    !Tr_meulage_motif_2 : Meulage d'un motif
    LOCAL CONST Robtarget Tr_meulage_motif_2_0 := [[50.49266796875,-116.5996484375,2.28227856445312],[0.000687502564593619,0.0161290141827085,0.042580986650659,-0.998962582791555],[0,0,0,0],[8.999999E+09,8.999999E+09,8.999999E+09,8.999999E+09,8.999999E+09,8.999999E+09]];
    LOCAL CONST Robtarget Tr_meulage_motif_2_1 := [[51.49176171875,-116.5571171875,2.28183227539063],[0.000687502564593619,0.0161290141827085,0.042580986650659,-0.998962582791555],[0,0,0,0],[8.999999E+09,8.999999E+09,8.999999E+09,8.999999E+09,8.999999E+09,8.999999E+09]];
    LOCAL CONST Robtarget Tr_meulage_motif_2_2 := [[52.490859375,-116.5145859375,2.2813857421875],[0.000687502564593619,0.0161290141827085,0.042580986650659,-0.998962582791555],[0,0,0,0],[8.999999E+09,8.999999E+09,8.999999E+09,8.999999E+09,8.999999E+09,8.999999E+09]];
    LOCAL CONST Robtarget Tr_meulage_motif_2_3 := [[53.489953125,-116.4720546875,2.280939453125],[0.000687502564593619,0.0161290141827085,0.042580986650659,-0.998962582791555],[0,0,0,0],[8.999999E+09,8.999999E+09,8.999999E+09,8.999999E+09,8.999999E+09,8.999999E+09]];
    LOCAL CONST Robtarget Tr_meulage_motif_2_4 := [[54.489046875,-116.4295234375,2.2804931640625],[0.000687502564593619,0.0161290141827085,0.042580986650659,-0.998962582791555],[0,0,0,0],[8.999999E+09,8.999999E+09,8.999999E+09,8.999999E+09,8.999999E+09,8.999999E+09]];
    LOCAL CONST Robtarget Tr_meulage_motif_2_5 := [[55.48814453125,-116.3869921875,2.28004663085937],[0.000687502564593619,0.0161290141827085,0.042580986650659,-0.998962582791555],[0,0,0,0],[8.999999E+09,8.999999E+09,8.999999E+09,8.999999E+09,8.999999E+09,8.999999E+09]];
    LOCAL CONST Robtarget Tr_meulage_motif_2_6 := [[56.48723828125,-116.3444609375,2.27960034179688],[0.000687502564593619,0.0161290141827085,0.042580986650659,-0.998962582791555],[0,0,0,0],[8.999999E+09,8.999999E+09,8.999999E+09,8.999999E+09,8.999999E+09,8.999999E+09]];
    LOCAL CONST Robtarget Tr_meulage_motif_2_7 := [[57.48633203125,-116.3019296875,2.27915405273438],[0.000687502564593619,0.0161290141827085,0.042580986650659,-0.998962582791555],[0,0,0,0],[8.999999E+09,8.999999E+09,8.999999E+09,8.999999E+09,8.999999E+09,8.999999E+09]];
    LOCAL CONST Robtarget Tr_meulage_motif_2_8 := [[58.4854296875,-116.2593984375,2.27870776367187],[0.000687502564593619,0.0161290141827085,0.042580986650659,-0.998962582791555],[0,0,0,0],[8.999999E+09,8.999999E+09,8.999999E+09,8.999999E+09,8.999999E+09,8.999999E+09]];
    LOCAL CONST Robtarget Tr_meulage_motif_2_9 := [[59.4845234375,-116.2168671875,2.27826123046875],[0.000687502564593619,0.0161290141827085,0.042580986650659,-0.998962582791555],[0,0,0,0],[8.999999E+09,8.999999E+09,8.999999E+09,8.999999E+09,8.999999E+09,8.999999E+09]];
    LOCAL CONST Robtarget Tr_meulage_motif_2_10 := [[60.4836171875,-116.1743359375,2.27781494140625],[0.000687502564593619,0.0161290141827085,0.042580986650659,-0.998962582791555],[0,0,0,0],[8.999999E+09,8.999999E+09,8.999999E+09,8.999999E+09,8.999999E+09,8.999999E+09]];
    LOCAL CONST Robtarget Tr_meulage_motif_2_11 := [[61.48271484375,-116.1318046875,2.27736865234375],[0.000687502564593619,0.0161290141827085,0.042580986650659,-0.998962582791555],[0,0,0,0],[8.999999E+09,8.999999E+09,8.999999E+09,8.999999E+09,8.999999E+09,8.999999E+09]];
    LOCAL CONST Robtarget Tr_meulage_motif_2_12 := [[62.48180859375,-116.0892734375,2.27692211914063],[0.000687502564593619,0.0161290141827085,0.042580986650659,-0.998962582791555],[0,0,0,0],[8.999999E+09,8.999999E+09,8.999999E+09,8.999999E+09,8.999999E+09,8.999999E+09]];
    LOCAL CONST Robtarget Tr_meulage_motif_2_13 := [[63.48090234375,-116.0467421875,2.27647583007812],[0.000687502564593619,0.0161290141827085,0.042580986650659,-0.998962582791555],[0,0,0,0],[8.999999E+09,8.999999E+09,8.999999E+09,8.999999E+09,8.999999E+09,8.999999E+09]];
    LOCAL CONST Robtarget Tr_meulage_motif_2_14 := [[64.47999609375,-116.0042109375,2.27602954101563],[0.000687502564593619,0.0161290141827085,0.042580986650659,-0.998962582791555],[0,0,0,0],[8.999999E+09,8.999999E+09,8.999999E+09,8.999999E+09,8.999999E+09,8.999999E+09]];
    LOCAL CONST Robtarget Tr_meulage_motif_2_15 := [[65.47909375,-115.9616796875,2.2755830078125],[0.000687502564593619,0.0161290141827085,0.042580986650659,-0.998962582791555],[0,0,0,0],[8.999999E+09,8.999999E+09,8.999999E+09,8.999999E+09,8.999999E+09,8.999999E+09]];
    LOCAL CONST Robtarget Tr_meulage_motif_2_16 := [[66.4781875,-115.9191484375,2.27513671875],[0.000687502564593619,0.0161290141827085,0.042580986650659,-0.998962582791555],[0,0,0,0],[8.999999E+09,8.999999E+09,8.999999E+09,8.999999E+09,8.999999E+09,8.999999E+09]];
    LOCAL CONST Robtarget Tr_meulage_motif_2_17 := [[67.47728125,-115.8766171875,2.2746904296875],[0.000687502564593619,0.0161290141827085,0.042580986650659,-0.998962582791555],[0,0,0,0],[8.999999E+09,8.999999E+09,8.999999E+09,8.999999E+09,8.999999E+09,8.999999E+09]];
    LOCAL CONST Robtarget Tr_meulage_motif_2_18 := [[68.476375,-115.8340859375,2.274244140625],[0.000687502564593619,0.0161290141827085,0.042580986650659,-0.998962582791555],[0,0,0,0],[8.999999E+09,8.999999E+09,8.999999E+09,8.999999E+09,8.999999E+09,8.999999E+09]];
    LOCAL CONST Robtarget Tr_meulage_motif_2_19 := [[69.4754765625,-115.7915546875,2.27379760742188],[0.000687502564593619,0.0161290141827085,0.042580986650659,-0.998962582791555],[0,0,0,0],[8.999999E+09,8.999999E+09,8.999999E+09,8.999999E+09,8.999999E+09,8.999999E+09]];
    LOCAL CONST Robtarget Tr_meulage_motif_2_20 := [[70.4745703125,-115.7490234375,2.27335131835938],[0.000687502564593619,0.0161290141827085,0.042580986650659,-0.998962582791555],[0,0,0,0],[8.999999E+09,8.999999E+09,8.999999E+09,8.999999E+09,8.999999E+09,8.999999E+09]];
    LOCAL CONST Robtarget Tr_meulage_motif_2_21 := [[71.4736640625,-115.7064921875,2.27290502929687],[0.000687502564593619,0.0161290141827085,0.042580986650659,-0.998962582791555],[0,0,0,0],[8.999999E+09,8.999999E+09,8.999999E+09,8.999999E+09,8.999999E+09,8.999999E+09]];
    LOCAL CONST Robtarget Tr_meulage_motif_2_22 := [[72.4727578125,-115.663953125,2.27245849609375],[0.000687502564593619,0.0161290141827085,0.042580986650659,-0.998962582791555],[0,0,0,0],[8.999999E+09,8.999999E+09,8.999999E+09,8.999999E+09,8.999999E+09,8.999999E+09]];
    LOCAL CONST Robtarget Tr_meulage_motif_2_23 := [[73.4718515625,-115.621421875,2.27201220703125],[0.000687502564593619,0.0161290141827085,0.042580986650659,-0.998962582791555],[0,0,0,0],[8.999999E+09,8.999999E+09,8.999999E+09,8.999999E+09,8.999999E+09,8.999999E+09]];
    LOCAL CONST Robtarget Tr_meulage_motif_2_24 := [[74.4709453125,-115.578890625,2.27156591796875],[0.000687502564593619,0.0161290141827085,0.042580986650659,-0.998962582791555],[0,0,0,0],[8.999999E+09,8.999999E+09,8.999999E+09,8.999999E+09,8.999999E+09,8.999999E+09]];
    LOCAL CONST Robtarget Tr_meulage_motif_2_25 := [[75.470046875,-115.536359375,2.27111938476563],[0.000687502564593619,0.0161290141827085,0.042580986650659,-0.998962582791555],[0,0,0,0],[8.999999E+09,8.999999E+09,8.999999E+09,8.999999E+09,8.999999E+09,8.999999E+09]];
    LOCAL CONST Robtarget Tr_meulage_motif_2_26 := [[76.469140625,-115.493828125,2.27067309570312],[0.000687502564593619,0.0161290141827085,0.042580986650659,-0.998962582791555],[0,0,0,0],[8.999999E+09,8.999999E+09,8.999999E+09,8.999999E+09,8.999999E+09,8.999999E+09]];
    LOCAL CONST Robtarget Tr_meulage_motif_2_27 := [[77.468234375,-115.451296875,2.27022680664063],[0.000687502564593619,0.0161290141827085,0.042580986650659,-0.998962582791555],[0,0,0,0],[8.999999E+09,8.999999E+09,8.999999E+09,8.999999E+09,8.999999E+09,8.999999E+09]];
    LOCAL CONST Robtarget Tr_meulage_motif_2_28 := [[78.467328125,-115.408765625,2.26978051757813],[0.000687502564593619,0.0161290141827085,0.042580986650659,-0.998962582791555],[0,0,0,0],[8.999999E+09,8.999999E+09,8.999999E+09,8.999999E+09,8.999999E+09,8.999999E+09]];
    LOCAL CONST Robtarget Tr_meulage_motif_2_29 := [[79.466421875,-115.366234375,2.269333984375],[0.000687502564593619,0.0161290141827085,0.042580986650659,-0.998962582791555],[0,0,0,0],[8.999999E+09,8.999999E+09,8.999999E+09,8.999999E+09,8.999999E+09,8.999999E+09]];
    LOCAL CONST Robtarget Tr_meulage_motif_2_30 := [[80.465515625,-115.323703125,2.2688876953125],[0.000687502564593619,0.0161290141827085,0.042580986650659,-0.998962582791555],[0,0,0,0],[8.999999E+09,8.999999E+09,8.999999E+09,8.999999E+09,8.999999E+09,8.999999E+09]];
    LOCAL CONST Robtarget Tr_meulage_motif_2_31 := [[81.4646171875,-115.281171875,2.26844140625],[0.000687502564593619,0.0161290141827085,0.042580986650659,-0.998962582791555],[0,0,0,0],[8.999999E+09,8.999999E+09,8.999999E+09,8.999999E+09,8.999999E+09,8.999999E+09]];
    LOCAL CONST Robtarget Tr_meulage_motif_2_32 := [[82.4637109375,-115.238640625,2.26799487304688],[0.000687502564593619,0.0161290141827085,0.042580986650659,-0.998962582791555],[0,0,0,0],[8.999999E+09,8.999999E+09,8.999999E+09,8.999999E+09,8.999999E+09,8.999999E+09]];
    LOCAL CONST Robtarget Tr_meulage_motif_2_33 := [[83.4628046875,-115.196109375,2.26754858398438],[0.000687502564593619,0.0161290141827085,0.042580986650659,-0.998962582791555],[0,0,0,0],[8.999999E+09,8.999999E+09,8.999999E+09,8.999999E+09,8.999999E+09,8.999999E+09]];
    LOCAL CONST Robtarget Tr_meulage_motif_2_34 := [[84.4618984375,-115.153578125,2.26710229492187],[0.000687502564593619,0.0161290141827085,0.042580986650659,-0.998962582791555],[0,0,0,0],[8.999999E+09,8.999999E+09,8.999999E+09,8.999999E+09,8.999999E+09,8.999999E+09]];
    LOCAL CONST Robtarget Tr_meulage_motif_2_35 := [[85.4609921875,-115.111046875,2.26665576171875],[0.000687502564593619,0.0161290141827085,0.042580986650659,-0.998962582791555],[0,0,0,0],[8.999999E+09,8.999999E+09,8.999999E+09,8.999999E+09,8.999999E+09,8.999999E+09]];
    LOCAL CONST Robtarget Tr_meulage_motif_2_36 := [[86.4600859375,-115.068515625,2.26620947265625],[0.000687502564593619,0.0161290141827085,0.042580986650659,-0.998962582791555],[0,0,0,0],[8.999999E+09,8.999999E+09,8.999999E+09,8.999999E+09,8.999999E+09,8.999999E+09]];
    LOCAL CONST Robtarget Tr_meulage_motif_2_37 := [[87.4591875,-115.025984375,2.26576318359375],[0.000687502564593619,0.0161290141827085,0.042580986650659,-0.998962582791555],[0,0,0,0],[8.999999E+09,8.999999E+09,8.999999E+09,8.999999E+09,8.999999E+09,8.999999E+09]];
    LOCAL CONST Robtarget Tr_meulage_motif_2_38 := [[88.45828125,-114.983453125,2.26531689453125],[0.000687502564593619,0.0161290141827085,0.042580986650659,-0.998962582791555],[0,0,0,0],[8.999999E+09,8.999999E+09,8.999999E+09,8.999999E+09,8.999999E+09,8.999999E+09]];
    LOCAL CONST Robtarget Tr_meulage_motif_2_39 := [[89.4452421875,-114.83075,2.26370166015625],[0.000687502564593619,0.0161290141827085,0.042580986650659,-0.998962582791555],[0,0,0,0],[8.999999E+09,8.999999E+09,8.999999E+09,8.999999E+09,8.999999E+09,8.999999E+09]];
    LOCAL CONST Robtarget Tr_meulage_motif_2_40 := [[90.3818984375,-114.5795078125,2.26104125976563],[0.000687502564593619,0.0161290141827085,0.042580986650659,-0.998962582791555],[0,0,0,0],[8.999999E+09,8.999999E+09,8.999999E+09,8.999999E+09,8.999999E+09,8.999999E+09]];
    LOCAL CONST Robtarget Tr_meulage_motif_2_41 := [[91.22228125,-114.2716640625,2.25777978515625],[0.000687502564593619,0.0161290141827085,0.042580986650659,-0.998962582791555],[0,0,0,0],[8.999999E+09,8.999999E+09,8.999999E+09,8.999999E+09,8.999999E+09,8.999999E+09]];
    LOCAL CONST Robtarget Tr_meulage_motif_2_42 := [[91.9598046875,-113.96409375,2.25452075195312],[0.000687502564593619,0.0161290141827085,0.042580986650659,-0.998962582791555],[0,0,0,0],[8.999999E+09,8.999999E+09,8.999999E+09,8.999999E+09,8.999999E+09,8.999999E+09]];
    LOCAL CONST Robtarget Tr_meulage_motif_2_43 := [[93.0336640625,-113.3017265625,2.2475],[0.000687502564593619,0.0161290141827085,0.042580986650659,-0.998962582791555],[0,0,0,0],[8.999999E+09,8.999999E+09,8.999999E+09,8.999999E+09,8.999999E+09,8.999999E+09]];
    LOCAL CONST Robtarget Tr_meulage_motif_2_44 := [[94.0205625,-112.41134375,2.23805981445313],[0.000687502564593619,0.0161290141827085,0.042580986650659,-0.998962582791555],[0,0,0,0],[8.999999E+09,8.999999E+09,8.999999E+09,8.999999E+09,8.999999E+09,8.999999E+09]];
    LOCAL CONST Robtarget Tr_meulage_motif_2_45 := [[94.8238984375,-111.3523984375,2.2268310546875],[0.000687502564593619,0.0161290141827085,0.042580986650659,-0.998962582791555],[0,0,0,0],[8.999999E+09,8.999999E+09,8.999999E+09,8.999999E+09,8.999999E+09,8.999999E+09]];
    LOCAL CONST Robtarget Tr_meulage_motif_2_46 := [[95.264140625,-110.2165234375,2.21478442382812],[0.000687502564593619,0.0161290141827085,0.042580986650659,-0.998962582791555],[0,0,0,0],[8.999999E+09,8.999999E+09,8.999999E+09,8.999999E+09,8.999999E+09,8.999999E+09]];
    LOCAL CONST Robtarget Tr_meulage_motif_2_47 := [[95.261578125,-109.5200703125,2.20739672851562],[0.000687502564593619,0.0161290141827085,0.042580986650659,-0.998962582791555],[0,0,0,0],[8.999999E+09,8.999999E+09,8.999999E+09,8.999999E+09,8.999999E+09,8.999999E+09]];
    LOCAL CONST Robtarget Tr_meulage_motif_2_48 := [[95.233453125,-108.8594609375,2.20038916015625],[0.000687502564593619,0.0161290141827085,0.042580986650659,-0.998962582791555],[0,0,0,0],[8.999999E+09,8.999999E+09,8.999999E+09,8.999999E+09,8.999999E+09,8.999999E+09]];
    LOCAL CONST Robtarget Tr_meulage_motif_2_49 := [[95.1505078125,-108.2013359375,2.19340771484375],[0.000687502564593619,0.0161290141827085,0.042580986650659,-0.998962582791555],[0,0,0,0],[8.999999E+09,8.999999E+09,8.999999E+09,8.999999E+09,8.999999E+09,8.999999E+09]];
    LOCAL CONST Robtarget Tr_meulage_motif_2_50 := [[94.605875,-107.121828125,2.18195434570312],[0.000687502564593619,0.0161290141827085,0.042580986650659,-0.998962582791555],[0,0,0,0],[8.999999E+09,8.999999E+09,8.999999E+09,8.999999E+09,8.999999E+09,8.999999E+09]];
    LOCAL CONST Robtarget Tr_meulage_motif_2_51 := [[93.7072109375,-106.152609375,2.17166918945313],[0.000687502564593619,0.0161290141827085,0.042580986650659,-0.998962582791555],[0,0,0,0],[8.999999E+09,8.999999E+09,8.999999E+09,8.999999E+09,8.999999E+09,8.999999E+09]];
    LOCAL CONST Robtarget Tr_meulage_motif_2_52 := [[92.6494765625,-105.3680546875,2.16334204101563],[0.000687502564593619,0.0161290141827085,0.042580986650659,-0.998962582791555],[0,0,0,0],[8.999999E+09,8.999999E+09,8.999999E+09,8.999999E+09,8.999999E+09,8.999999E+09]];
    LOCAL CONST Robtarget Tr_meulage_motif_2_53 := [[91.946171875,-105.00190625,2.15945458984375],[0.000687502564593619,0.0161290141827085,0.042580986650659,-0.998962582791555],[0,0,0,0],[8.999999E+09,8.999999E+09,8.999999E+09,8.999999E+09,8.999999E+09,8.999999E+09]];
    LOCAL CONST Robtarget Tr_meulage_motif_2_54 := [[90.768328125,-104.5641015625,2.15480517578125],[0.000687502564593619,0.0161290141827085,0.042580986650659,-0.998962582791555],[0,0,0,0],[8.999999E+09,8.999999E+09,8.999999E+09,8.999999E+09,8.999999E+09,8.999999E+09]];
    LOCAL CONST Robtarget Tr_meulage_motif_2_55 := [[89.912828125,-104.336203125,2.15238354492188],[0.000687502564593619,0.0161290141827085,0.042580986650659,-0.998962582791555],[0,0,0,0],[8.999999E+09,8.999999E+09,8.999999E+09,8.999999E+09,8.999999E+09,8.999999E+09]];
    LOCAL CONST Robtarget Tr_meulage_motif_2_56 := [[88.9729765625,-104.1715703125,2.1506328125],[0.000687502564593619,0.0161290141827085,0.042580986650659,-0.998962582791555],[0,0,0,0],[8.999999E+09,8.999999E+09,8.999999E+09,8.999999E+09,8.999999E+09,8.999999E+09]];
    LOCAL CONST Robtarget Tr_meulage_motif_2_57 := [[87.9876796875,-104.104828125,2.149919921875],[0.000687502564593619,0.0161290141827085,0.042580986650659,-0.998962582791555],[0,0,0,0],[8.999999E+09,8.999999E+09,8.999999E+09,8.999999E+09,8.999999E+09,8.999999E+09]];
    LOCAL CONST Robtarget Tr_meulage_motif_2_58 := [[86.9913125,-104.0365546875,2.14919091796875],[0.000687502564593619,0.0161290141827085,0.042580986650659,-0.998962582791555],[0,0,0,0],[8.999999E+09,8.999999E+09,8.999999E+09,8.999999E+09,8.999999E+09,8.999999E+09]];
    LOCAL CONST Robtarget Tr_meulage_motif_2_59 := [[85.99221875,-104.0790859375,2.14963745117188],[0.000687502564593619,0.0161290141827085,0.042580986650659,-0.998962582791555],[0,0,0,0],[8.999999E+09,8.999999E+09,8.999999E+09,8.999999E+09,8.999999E+09,8.999999E+09]];
    LOCAL CONST Robtarget Tr_meulage_motif_2_60 := [[84.993125,-104.121625,2.15008374023438],[0.000687502564593619,0.0161290141827085,0.042580986650659,-0.998962582791555],[0,0,0,0],[8.999999E+09,8.999999E+09,8.999999E+09,8.999999E+09,8.999999E+09,8.999999E+09]];
    LOCAL CONST Robtarget Tr_meulage_motif_2_61 := [[83.9940234375,-104.16415625,2.15053002929687],[0.000687502564593619,0.0161290141827085,0.042580986650659,-0.998962582791555],[0,0,0,0],[8.999999E+09,8.999999E+09,8.999999E+09,8.999999E+09,8.999999E+09,8.999999E+09]];
    LOCAL CONST Robtarget Tr_meulage_motif_2_62 := [[82.9949296875,-104.2066875,2.1509765625],[0.000687502564593619,0.0161290141827085,0.042580986650659,-0.998962582791555],[0,0,0,0],[8.999999E+09,8.999999E+09,8.999999E+09,8.999999E+09,8.999999E+09,8.999999E+09]];
    LOCAL CONST Robtarget Tr_meulage_motif_2_63 := [[81.9958359375,-104.24921875,2.1514228515625],[0.000687502564593619,0.0161290141827085,0.042580986650659,-0.998962582791555],[0,0,0,0],[8.999999E+09,8.999999E+09,8.999999E+09,8.999999E+09,8.999999E+09,8.999999E+09]];
    LOCAL CONST Robtarget Tr_meulage_motif_2_64 := [[80.9967421875,-104.29175,2.151869140625],[0.000687502564593619,0.0161290141827085,0.042580986650659,-0.998962582791555],[0,0,0,0],[8.999999E+09,8.999999E+09,8.999999E+09,8.999999E+09,8.999999E+09,8.999999E+09]];
    LOCAL CONST Robtarget Tr_meulage_motif_2_65 := [[79.9976484375,-104.33428125,2.15231567382813],[0.000687502564593619,0.0161290141827085,0.042580986650659,-0.998962582791555],[0,0,0,0],[8.999999E+09,8.999999E+09,8.999999E+09,8.999999E+09,8.999999E+09,8.999999E+09]];
    LOCAL CONST Robtarget Tr_meulage_motif_2_66 := [[78.9985546875,-104.3768125,2.15276196289062],[0.000687502564593619,0.0161290141827085,0.042580986650659,-0.998962582791555],[0,0,0,0],[8.999999E+09,8.999999E+09,8.999999E+09,8.999999E+09,8.999999E+09,8.999999E+09]];
    LOCAL CONST Robtarget Tr_meulage_motif_2_67 := [[77.999453125,-104.41934375,2.15320825195313],[0.000687502564593619,0.0161290141827085,0.042580986650659,-0.998962582791555],[0,0,0,0],[8.999999E+09,8.999999E+09,8.999999E+09,8.999999E+09,8.999999E+09,8.999999E+09]];
    LOCAL CONST Robtarget Tr_meulage_motif_2_68 := [[77.000359375,-104.461875,2.15365454101563],[0.000687502564593619,0.0161290141827085,0.042580986650659,-0.998962582791555],[0,0,0,0],[8.999999E+09,8.999999E+09,8.999999E+09,8.999999E+09,8.999999E+09,8.999999E+09]];
    LOCAL CONST Robtarget Tr_meulage_motif_2_69 := [[76.001265625,-104.50440625,2.15410107421875],[0.000687502564593619,0.0161290141827085,0.042580986650659,-0.998962582791555],[0,0,0,0],[8.999999E+09,8.999999E+09,8.999999E+09,8.999999E+09,8.999999E+09,8.999999E+09]];
    LOCAL CONST Robtarget Tr_meulage_motif_2_70 := [[75.002171875,-104.5469375,2.15454736328125],[0.000687502564593619,0.0161290141827085,0.042580986650659,-0.998962582791555],[0,0,0,0],[8.999999E+09,8.999999E+09,8.999999E+09,8.999999E+09,8.999999E+09,8.999999E+09]];
    LOCAL CONST Robtarget Tr_meulage_motif_2_71 := [[74.003078125,-104.58946875,2.15499365234375],[0.000687502564593619,0.0161290141827085,0.042580986650659,-0.998962582791555],[0,0,0,0],[8.999999E+09,8.999999E+09,8.999999E+09,8.999999E+09,8.999999E+09,8.999999E+09]];
    LOCAL CONST Robtarget Tr_meulage_motif_2_72 := [[73.003984375,-104.632,2.15544018554688],[0.000687502564593619,0.0161290141827085,0.042580986650659,-0.998962582791555],[0,0,0,0],[8.999999E+09,8.999999E+09,8.999999E+09,8.999999E+09,8.999999E+09,8.999999E+09]];
    LOCAL CONST Robtarget Tr_meulage_motif_2_73 := [[72.0048828125,-104.67453125,2.15588647460938],[0.000687502564593619,0.0161290141827085,0.042580986650659,-0.998962582791555],[0,0,0,0],[8.999999E+09,8.999999E+09,8.999999E+09,8.999999E+09,8.999999E+09,8.999999E+09]];
    LOCAL CONST Robtarget Tr_meulage_motif_2_74 := [[71.0057890625,-104.7170625,2.15633276367187],[0.000687502564593619,0.0161290141827085,0.042580986650659,-0.998962582791555],[0,0,0,0],[8.999999E+09,8.999999E+09,8.999999E+09,8.999999E+09,8.999999E+09,8.999999E+09]];
    LOCAL CONST Robtarget Tr_meulage_motif_2_75 := [[70.0066953125,-104.75959375,2.156779296875],[0.000687502564593619,0.0161290141827085,0.042580986650659,-0.998962582791555],[0,0,0,0],[8.999999E+09,8.999999E+09,8.999999E+09,8.999999E+09,8.999999E+09,8.999999E+09]];
    LOCAL CONST Robtarget Tr_meulage_motif_2_76 := [[69.0076015625,-104.802125,2.1572255859375],[0.000687502564593619,0.0161290141827085,0.042580986650659,-0.998962582791555],[0,0,0,0],[8.999999E+09,8.999999E+09,8.999999E+09,8.999999E+09,8.999999E+09,8.999999E+09]];
    LOCAL CONST Robtarget Tr_meulage_motif_2_77 := [[68.0085078125,-104.84465625,2.157671875],[0.000687502564593619,0.0161290141827085,0.042580986650659,-0.998962582791555],[0,0,0,0],[8.999999E+09,8.999999E+09,8.999999E+09,8.999999E+09,8.999999E+09,8.999999E+09]];
    LOCAL CONST Robtarget Tr_meulage_motif_2_78 := [[67.0094140625,-104.8871875,2.1581181640625],[0.000687502564593619,0.0161290141827085,0.042580986650659,-0.998962582791555],[0,0,0,0],[8.999999E+09,8.999999E+09,8.999999E+09,8.999999E+09,8.999999E+09,8.999999E+09]];
    LOCAL CONST Robtarget Tr_meulage_motif_2_79 := [[66.0103203125,-104.92971875,2.15856469726562],[0.000687502564593619,0.0161290141827085,0.042580986650659,-0.998962582791555],[0,0,0,0],[8.999999E+09,8.999999E+09,8.999999E+09,8.999999E+09,8.999999E+09,8.999999E+09]];
    LOCAL CONST Robtarget Tr_meulage_motif_2_80 := [[65.01122265625,-104.97225,2.15901098632812],[0.000687502564593619,0.0161290141827085,0.042580986650659,-0.998962582791555],[0,0,0,0],[8.999999E+09,8.999999E+09,8.999999E+09,8.999999E+09,8.999999E+09,8.999999E+09]];
    LOCAL CONST Robtarget Tr_meulage_motif_2_81 := [[64.012125,-105.01478125,2.15945727539063],[0.000687502564593619,0.0161290141827085,0.042580986650659,-0.998962582791555],[0,0,0,0],[8.999999E+09,8.999999E+09,8.999999E+09,8.999999E+09,8.999999E+09,8.999999E+09]];
    LOCAL CONST Robtarget Tr_meulage_motif_2_82 := [[63.01303125,-105.0573125,2.15990380859375],[0.000687502564593619,0.0161290141827085,0.042580986650659,-0.998962582791555],[0,0,0,0],[8.999999E+09,8.999999E+09,8.999999E+09,8.999999E+09,8.999999E+09,8.999999E+09]];
    LOCAL CONST Robtarget Tr_meulage_motif_2_83 := [[62.0139375,-105.09984375,2.16035009765625],[0.000687502564593619,0.0161290141827085,0.042580986650659,-0.998962582791555],[0,0,0,0],[8.999999E+09,8.999999E+09,8.999999E+09,8.999999E+09,8.999999E+09,8.999999E+09]];
    LOCAL CONST Robtarget Tr_meulage_motif_2_84 := [[61.01483984375,-105.142375,2.16079638671875],[0.000687502564593619,0.0161290141827085,0.042580986650659,-0.998962582791555],[0,0,0,0],[8.999999E+09,8.999999E+09,8.999999E+09,8.999999E+09,8.999999E+09,8.999999E+09]];
    LOCAL CONST Robtarget Tr_meulage_motif_2_85 := [[60.01574609375,-105.18490625,2.16124291992188],[0.000687502564593619,0.0161290141827085,0.042580986650659,-0.998962582791555],[0,0,0,0],[8.999999E+09,8.999999E+09,8.999999E+09,8.999999E+09,8.999999E+09,8.999999E+09]];
    LOCAL CONST Robtarget Tr_meulage_motif_2_86 := [[59.01665234375,-105.2274375,2.16168920898438],[0.000687502564593619,0.0161290141827085,0.042580986650659,-0.998962582791555],[0,0,0,0],[8.999999E+09,8.999999E+09,8.999999E+09,8.999999E+09,8.999999E+09,8.999999E+09]];
    LOCAL CONST Robtarget Tr_meulage_motif_2_87 := [[58.0175546875,-105.26996875,2.16213549804687],[0.000687502564593619,0.0161290141827085,0.042580986650659,-0.998962582791555],[0,0,0,0],[8.999999E+09,8.999999E+09,8.999999E+09,8.999999E+09,8.999999E+09,8.999999E+09]];
    LOCAL CONST Robtarget Tr_meulage_motif_2_88 := [[57.0184609375,-105.3125,2.16258178710937],[0.000687502564593619,0.0161290141827085,0.042580986650659,-0.998962582791555],[0,0,0,0],[8.999999E+09,8.999999E+09,8.999999E+09,8.999999E+09,8.999999E+09,8.999999E+09]];
    LOCAL CONST Robtarget Tr_meulage_motif_2_89 := [[56.02209375,-105.2442265625,2.16185302734375],[0.000687502564593619,0.0161290141827085,0.042580986650659,-0.998962582791555],[0,0,0,0],[8.999999E+09,8.999999E+09,8.999999E+09,8.999999E+09,8.999999E+09,8.999999E+09]];
    LOCAL CONST Robtarget Tr_meulage_motif_2_90 := [[55.06746875,-105.0735,2.16003735351563],[0.000687502564593619,0.0161290141827085,0.042580986650659,-0.998962582791555],[0,0,0,0],[8.999999E+09,8.999999E+09,8.999999E+09,8.999999E+09,8.999999E+09,8.999999E+09]];
    LOCAL CONST Robtarget Tr_meulage_motif_2_91 := [[54.20395703125,-104.8381875,2.157537109375],[0.000687502564593619,0.0161290141827085,0.042580986650659,-0.998962582791555],[0,0,0,0],[8.999999E+09,8.999999E+09,8.999999E+09,8.999999E+09,8.999999E+09,8.999999E+09]];
    LOCAL CONST Robtarget Tr_meulage_motif_2_92 := [[53.4801640625,-104.5645859375,2.15463134765625],[0.000687502564593619,0.0161290141827085,0.042580986650659,-0.998962582791555],[0,0,0,0],[8.999999E+09,8.999999E+09,8.999999E+09,8.999999E+09,8.999999E+09,8.999999E+09]];
    LOCAL CONST Robtarget Tr_meulage_motif_2_93 := [[52.418453125,-103.9466875,2.14807202148438],[0.000687502564593619,0.0161290141827085,0.042580986650659,-0.998962582791555],[0,0,0,0],[8.999999E+09,8.999999E+09,8.999999E+09,8.999999E+09,8.999999E+09,8.999999E+09]];
    LOCAL CONST Robtarget Tr_meulage_motif_2_94 := [[51.47896875,-103.0839765625,2.13891625976563],[0.000687502564593619,0.0161290141827085,0.042580986650659,-0.998962582791555],[0,0,0,0],[8.999999E+09,8.999999E+09,8.999999E+09,8.999999E+09,8.999999E+09,8.999999E+09]];
    LOCAL CONST Robtarget Tr_meulage_motif_2_95 := [[50.8999921875,-102.061703125,2.12806982421875],[0.000687502564593619,0.0161290141827085,0.042580986650659,-0.998962582791555],[0,0,0,0],[8.999999E+09,8.999999E+09,8.999999E+09,8.999999E+09,8.999999E+09,8.999999E+09]];
    LOCAL CONST Robtarget Tr_meulage_motif_2_96 := [[50.685890625,-101.3770078125,2.12080590820312],[0.000687502564593619,0.0161290141827085,0.042580986650659,-0.998962582791555],[0,0,0,0],[8.999999E+09,8.999999E+09,8.999999E+09,8.999999E+09,8.999999E+09,8.999999E+09]];
    LOCAL CONST Robtarget Tr_meulage_motif_2_97 := [[50.58935546875,-100.61046875,2.11267456054687],[0.000687502564593619,0.0161290141827085,0.042580986650659,-0.998962582791555],[0,0,0,0],[8.999999E+09,8.999999E+09,8.999999E+09,8.999999E+09,8.999999E+09,8.999999E+09]];
    LOCAL CONST Robtarget Tr_meulage_motif_2_98 := [[50.62348828125,-99.838484375,2.10448583984375],[0.000687502564593619,0.0161290141827085,0.042580986650659,-0.998962582791555],[0,0,0,0],[8.999999E+09,8.999999E+09,8.999999E+09,8.999999E+09,8.999999E+09,8.999999E+09]];
    LOCAL CONST Robtarget Tr_meulage_motif_2_99 := [[50.9955625,-98.713453125,2.09255395507813],[0.000687502564593619,0.0161290141827085,0.042580986650659,-0.998962582791555],[0,0,0,0],[8.999999E+09,8.999999E+09,8.999999E+09,8.999999E+09,8.999999E+09,8.999999E+09]];
    LOCAL CONST Robtarget Tr_meulage_motif_2_100 := [[51.38458984375,-98.110703125,2.086162109375],[0.000687502564593619,0.0161290141827085,0.042580986650659,-0.998962582791555],[0,0,0,0],[8.999999E+09,8.999999E+09,8.999999E+09,8.999999E+09,8.999999E+09,8.999999E+09]];
    LOCAL CONST Robtarget Tr_meulage_motif_2_101 := [[52.2331796875,-97.186703125,2.07636499023438],[0.000687502564593619,0.0161290141827085,0.042580986650659,-0.998962582791555],[0,0,0,0],[8.999999E+09,8.999999E+09,8.999999E+09,8.999999E+09,8.999999E+09,8.999999E+09]];
    LOCAL CONST Robtarget Tr_meulage_motif_2_102 := [[52.80071484375,-96.7478828125,2.071712890625],[0.000687502564593619,0.0161290141827085,0.042580986650659,-0.998962582791555],[0,0,0,0],[8.999999E+09,8.999999E+09,8.999999E+09,8.999999E+09,8.999999E+09,8.999999E+09]];
    LOCAL CONST Robtarget Tr_meulage_motif_2_103 := [[53.89446484375,-96.156765625,2.06544775390625],[0.000687502564593619,0.0161290141827085,0.042580986650659,-0.998962582791555],[0,0,0,0],[8.999999E+09,8.999999E+09,8.999999E+09,8.999999E+09,8.999999E+09,8.999999E+09]];
    LOCAL CONST Robtarget Tr_meulage_motif_2_104 := [[54.7067421875,-95.8264296875,2.06194775390625],[0.000687502564593619,0.0161290141827085,0.042580986650659,-0.998962582791555],[0,0,0,0],[8.999999E+09,8.999999E+09,8.999999E+09,8.999999E+09,8.999999E+09,8.999999E+09]];
    LOCAL CONST Robtarget Tr_meulage_motif_2_105 := [[55.629203125,-95.5825234375,2.05936499023437],[0.000687502564593619,0.0161290141827085,0.042580986650659,-0.998962582791555],[0,0,0,0],[8.999999E+09,8.999999E+09,8.999999E+09,8.999999E+09,8.999999E+09,8.999999E+09]];
    LOCAL CONST Robtarget Tr_meulage_motif_2_106 := [[56.6052578125,-95.43228125,2.05777587890625],[0.000687502564593619,0.0161290141827085,0.042580986650659,-0.998962582791555],[0,0,0,0],[8.999999E+09,8.999999E+09,8.999999E+09,8.999999E+09,8.999999E+09,8.999999E+09]];
    LOCAL CONST Robtarget Tr_meulage_motif_2_107 := [[57.59221875,-95.279578125,2.05616088867187],[0.000687502564593619,0.0161290141827085,0.042580986650659,-0.998962582791555],[0,0,0,0],[8.999999E+09,8.999999E+09,8.999999E+09,8.999999E+09,8.999999E+09,8.999999E+09]];
    LOCAL CONST Robtarget Tr_meulage_motif_2_108 := [[58.5913125,-95.237046875,2.05571459960938],[0.000687502564593619,0.0161290141827085,0.042580986650659,-0.998962582791555],[0,0,0,0],[8.999999E+09,8.999999E+09,8.999999E+09,8.999999E+09,8.999999E+09,8.999999E+09]];
    LOCAL CONST Robtarget Tr_meulage_motif_2_109 := [[59.59041015625,-95.194515625,2.05526806640625],[0.000687502564593619,0.0161290141827085,0.042580986650659,-0.998962582791555],[0,0,0,0],[8.999999E+09,8.999999E+09,8.999999E+09,8.999999E+09,8.999999E+09,8.999999E+09]];
    LOCAL CONST Robtarget Tr_meulage_motif_2_110 := [[60.58950390625,-95.151984375,2.05482177734375],[0.000687502564593619,0.0161290141827085,0.042580986650659,-0.998962582791555],[0,0,0,0],[8.999999E+09,8.999999E+09,8.999999E+09,8.999999E+09,8.999999E+09,8.999999E+09]];
    LOCAL CONST Robtarget Tr_meulage_motif_2_111 := [[61.58859765625,-95.109453125,2.05437548828125],[0.000687502564593619,0.0161290141827085,0.042580986650659,-0.998962582791555],[0,0,0,0],[8.999999E+09,8.999999E+09,8.999999E+09,8.999999E+09,8.999999E+09,8.999999E+09]];
    LOCAL CONST Robtarget Tr_meulage_motif_2_112 := [[62.5876953125,-95.066921875,2.05392919921875],[0.000687502564593619,0.0161290141827085,0.042580986650659,-0.998962582791555],[0,0,0,0],[8.999999E+09,8.999999E+09,8.999999E+09,8.999999E+09,8.999999E+09,8.999999E+09]];
    LOCAL CONST Robtarget Tr_meulage_motif_2_113 := [[63.5867890625,-95.024390625,2.05348266601563],[0.000687502564593619,0.0161290141827085,0.042580986650659,-0.998962582791555],[0,0,0,0],[8.999999E+09,8.999999E+09,8.999999E+09,8.999999E+09,8.999999E+09,8.999999E+09]];
    LOCAL CONST Robtarget Tr_meulage_motif_2_114 := [[64.5858828125,-94.981859375,2.05303637695313],[0.000687502564593619,0.0161290141827085,0.042580986650659,-0.998962582791555],[0,0,0,0],[8.999999E+09,8.999999E+09,8.999999E+09,8.999999E+09,8.999999E+09,8.999999E+09]];
    LOCAL CONST Robtarget Tr_meulage_motif_2_115 := [[65.5849765625,-94.939328125,2.05259008789062],[0.000687502564593619,0.0161290141827085,0.042580986650659,-0.998962582791555],[0,0,0,0],[8.999999E+09,8.999999E+09,8.999999E+09,8.999999E+09,8.999999E+09,8.999999E+09]];
    LOCAL CONST Robtarget Tr_meulage_motif_2_116 := [[66.5840703125,-94.896796875,2.0521435546875],[0.000687502564593619,0.0161290141827085,0.042580986650659,-0.998962582791555],[0,0,0,0],[8.999999E+09,8.999999E+09,8.999999E+09,8.999999E+09,8.999999E+09,8.999999E+09]];
    LOCAL CONST Robtarget Tr_meulage_motif_2_117 := [[67.583171875,-94.854265625,2.051697265625],[0.000687502564593619,0.0161290141827085,0.042580986650659,-0.998962582791555],[0,0,0,0],[8.999999E+09,8.999999E+09,8.999999E+09,8.999999E+09,8.999999E+09,8.999999E+09]];
    LOCAL CONST Robtarget Tr_meulage_motif_2_118 := [[68.582265625,-94.811734375,2.0512509765625],[0.000687502564593619,0.0161290141827085,0.042580986650659,-0.998962582791555],[0,0,0,0],[8.999999E+09,8.999999E+09,8.999999E+09,8.999999E+09,8.999999E+09,8.999999E+09]];
    LOCAL CONST Robtarget Tr_meulage_motif_2_119 := [[69.581359375,-94.769203125,2.05080444335937],[0.000687502564593619,0.0161290141827085,0.042580986650659,-0.998962582791555],[0,0,0,0],[8.999999E+09,8.999999E+09,8.999999E+09,8.999999E+09,8.999999E+09,8.999999E+09]];
    LOCAL CONST Robtarget Tr_meulage_motif_2_120 := [[70.580453125,-94.726671875,2.05035815429687],[0.000687502564593619,0.0161290141827085,0.042580986650659,-0.998962582791555],[0,0,0,0],[8.999999E+09,8.999999E+09,8.999999E+09,8.999999E+09,8.999999E+09,8.999999E+09]];
    LOCAL CONST Robtarget Tr_meulage_motif_2_121 := [[71.579546875,-94.684140625,2.04991186523438],[0.000687502564593619,0.0161290141827085,0.042580986650659,-0.998962582791555],[0,0,0,0],[8.999999E+09,8.999999E+09,8.999999E+09,8.999999E+09,8.999999E+09,8.999999E+09]];
    LOCAL CONST Robtarget Tr_meulage_motif_2_122 := [[72.578640625,-94.641609375,2.04946557617188],[0.000687502564593619,0.0161290141827085,0.042580986650659,-0.998962582791555],[0,0,0,0],[8.999999E+09,8.999999E+09,8.999999E+09,8.999999E+09,8.999999E+09,8.999999E+09]];
    LOCAL CONST Robtarget Tr_meulage_motif_2_123 := [[73.5777421875,-94.599078125,2.04901904296875],[0.000687502564593619,0.0161290141827085,0.042580986650659,-0.998962582791555],[0,0,0,0],[8.999999E+09,8.999999E+09,8.999999E+09,8.999999E+09,8.999999E+09,8.999999E+09]];
    LOCAL CONST Robtarget Tr_meulage_motif_2_124 := [[74.5768359375,-94.556546875,2.04857275390625],[0.000687502564593619,0.0161290141827085,0.042580986650659,-0.998962582791555],[0,0,0,0],[8.999999E+09,8.999999E+09,8.999999E+09,8.999999E+09,8.999999E+09,8.999999E+09]];
    LOCAL CONST Robtarget Tr_meulage_motif_2_125 := [[75.5759296875,-94.514015625,2.04812646484375],[0.000687502564593619,0.0161290141827085,0.042580986650659,-0.998962582791555],[0,0,0,0],[8.999999E+09,8.999999E+09,8.999999E+09,8.999999E+09,8.999999E+09,8.999999E+09]];
    LOCAL CONST Robtarget Tr_meulage_motif_2_126 := [[76.5750234375,-94.471484375,2.04768005371094],[0.000687502564593619,0.0161290141827085,0.042580986650659,-0.998962582791555],[0,0,0,0],[8.999999E+09,8.999999E+09,8.999999E+09,8.999999E+09,8.999999E+09,8.999999E+09]];
    LOCAL CONST Robtarget Tr_meulage_motif_2_127 := [[77.5741171875,-94.428953125,2.04723364257813],[0.000687502564593619,0.0161290141827085,0.042580986650659,-0.998962582791555],[0,0,0,0],[8.999999E+09,8.999999E+09,8.999999E+09,8.999999E+09,8.999999E+09,8.999999E+09]];
    LOCAL CONST Robtarget Tr_meulage_motif_2_128 := [[78.5732109375,-94.386421875,2.04678735351562],[0.000687502564593619,0.0161290141827085,0.042580986650659,-0.998962582791555],[0,0,0,0],[8.999999E+09,8.999999E+09,8.999999E+09,8.999999E+09,8.999999E+09,8.999999E+09]];
    LOCAL CONST Robtarget Tr_meulage_motif_2_129 := [[79.5723125,-94.343890625,2.04634094238281],[0.000687502564593619,0.0161290141827085,0.042580986650659,-0.998962582791555],[0,0,0,0],[8.999999E+09,8.999999E+09,8.999999E+09,8.999999E+09,8.999999E+09,8.999999E+09]];
    LOCAL CONST Robtarget Tr_meulage_motif_2_130 := [[80.57140625,-94.301359375,2.04589453125],[0.000687502564593619,0.0161290141827085,0.042580986650659,-0.998962582791555],[0,0,0,0],[8.999999E+09,8.999999E+09,8.999999E+09,8.999999E+09,8.999999E+09,8.999999E+09]];
    LOCAL CONST Robtarget Tr_meulage_motif_2_131 := [[81.5705,-94.258828125,2.0454482421875],[0.000687502564593619,0.0161290141827085,0.042580986650659,-0.998962582791555],[0,0,0,0],[8.999999E+09,8.999999E+09,8.999999E+09,8.999999E+09,8.999999E+09,8.999999E+09]];
    LOCAL CONST Robtarget Tr_meulage_motif_2_132 := [[82.56959375,-94.216296875,2.04500183105469],[0.000687502564593619,0.0161290141827085,0.042580986650659,-0.998962582791555],[0,0,0,0],[8.999999E+09,8.999999E+09,8.999999E+09,8.999999E+09,8.999999E+09,8.999999E+09]];
    LOCAL CONST Robtarget Tr_meulage_motif_2_133 := [[83.5686875,-94.173765625,2.04455554199219],[0.000687502564593619,0.0161290141827085,0.042580986650659,-0.998962582791555],[0,0,0,0],[8.999999E+09,8.999999E+09,8.999999E+09,8.999999E+09,8.999999E+09,8.999999E+09]];
    LOCAL CONST Robtarget Tr_meulage_motif_2_134 := [[84.56778125,-94.131234375,2.04410913085938],[0.000687502564593619,0.0161290141827085,0.042580986650659,-0.998962582791555],[0,0,0,0],[8.999999E+09,8.999999E+09,8.999999E+09,8.999999E+09,8.999999E+09,8.999999E+09]];
    LOCAL CONST Robtarget Tr_meulage_motif_2_135 := [[85.5668828125,-94.088703125,2.04366271972656],[0.000687502564593619,0.0161290141827085,0.042580986650659,-0.998962582791555],[0,0,0,0],[8.999999E+09,8.999999E+09,8.999999E+09,8.999999E+09,8.999999E+09,8.999999E+09]];
    LOCAL CONST Robtarget Tr_meulage_motif_2_136 := [[86.5659765625,-94.046171875,2.04321643066406],[0.000687502564593619,0.0161290141827085,0.042580986650659,-0.998962582791555],[0,0,0,0],[8.999999E+09,8.999999E+09,8.999999E+09,8.999999E+09,8.999999E+09,8.999999E+09]];
    LOCAL CONST Robtarget Tr_meulage_motif_2_137 := [[87.5650703125,-94.003640625,2.04277001953125],[0.000687502564593619,0.0161290141827085,0.042580986650659,-0.998962582791555],[0,0,0,0],[8.999999E+09,8.999999E+09,8.999999E+09,8.999999E+09,8.999999E+09,8.999999E+09]];
    LOCAL CONST Robtarget Tr_meulage_motif_2_138 := [[88.55203125,-93.8509375,2.04115502929687],[0.000687502564593619,0.0161290141827085,0.042580986650659,-0.998962582791555],[0,0,0,0],[8.999999E+09,8.999999E+09,8.999999E+09,8.999999E+09,8.999999E+09,8.999999E+09]];
    LOCAL CONST Robtarget Tr_meulage_motif_2_139 := [[89.4886875,-93.5996953125,2.03849438476563],[0.000687502564593619,0.0161290141827085,0.042580986650659,-0.998962582791555],[0,0,0,0],[8.999999E+09,8.999999E+09,8.999999E+09,8.999999E+09,8.999999E+09,8.999999E+09]];
    LOCAL CONST Robtarget Tr_meulage_motif_2_140 := [[90.329078125,-93.29184375,2.03523291015625],[0.000687502564593619,0.0161290141827085,0.042580986650659,-0.998962582791555],[0,0,0,0],[8.999999E+09,8.999999E+09,8.999999E+09,8.999999E+09,8.999999E+09,8.999999E+09]];
    LOCAL CONST Robtarget Tr_meulage_motif_2_141 := [[91.06659375,-92.98428125,2.03197399902344],[0.000687502564593619,0.0161290141827085,0.042580986650659,-0.998962582791555],[0,0,0,0],[8.999999E+09,8.999999E+09,8.999999E+09,8.999999E+09,8.999999E+09,8.999999E+09]];
    LOCAL CONST Robtarget Tr_meulage_motif_2_142 := [[92.1404609375,-92.3219140625,2.024953125],[0.000687502564593619,0.0161290141827085,0.042580986650659,-0.998962582791555],[0,0,0,0],[8.999999E+09,8.999999E+09,8.999999E+09,8.999999E+09,8.999999E+09,8.999999E+09]];
    LOCAL CONST Robtarget Tr_meulage_motif_2_143 := [[93.1273515625,-91.4315234375,2.01551318359375],[0.000687502564593619,0.0161290141827085,0.042580986650659,-0.998962582791555],[0,0,0,0],[8.999999E+09,8.999999E+09,8.999999E+09,8.999999E+09,8.999999E+09,8.999999E+09]];
    LOCAL CONST Robtarget Tr_meulage_motif_2_144 := [[93.9306875,-90.3725859375,2.00428430175781],[0.000687502564593619,0.0161290141827085,0.042580986650659,-0.998962582791555],[0,0,0,0],[8.999999E+09,8.999999E+09,8.999999E+09,8.999999E+09,8.999999E+09,8.999999E+09]];
    LOCAL CONST Robtarget Tr_meulage_motif_2_145 := [[94.3709296875,-89.2367109375,1.99223767089844],[0.000687502564593619,0.0161290141827085,0.042580986650659,-0.998962582791555],[0,0,0,0],[8.999999E+09,8.999999E+09,8.999999E+09,8.999999E+09,8.999999E+09,8.999999E+09]];
    LOCAL CONST Robtarget Tr_meulage_motif_2_146 := [[94.3683671875,-88.5402578125,1.98485009765625],[0.000687502564593619,0.0161290141827085,0.042580986650659,-0.998962582791555],[0,0,0,0],[8.999999E+09,8.999999E+09,8.999999E+09,8.999999E+09,8.999999E+09,8.999999E+09]];
    LOCAL CONST Robtarget Tr_meulage_motif_2_147 := [[94.3402421875,-87.879640625,1.97784252929688],[0.000687502564593619,0.0161290141827085,0.042580986650659,-0.998962582791555],[0,0,0,0],[8.999999E+09,8.999999E+09,8.999999E+09,8.999999E+09,8.999999E+09,8.999999E+09]];
    LOCAL CONST Robtarget Tr_meulage_motif_2_148 := [[94.257296875,-87.221515625,1.97086108398437],[0.000687502564593619,0.0161290141827085,0.042580986650659,-0.998962582791555],[0,0,0,0],[8.999999E+09,8.999999E+09,8.999999E+09,8.999999E+09,8.999999E+09,8.999999E+09]];
    LOCAL CONST Robtarget Tr_meulage_motif_2_149 := [[93.7126640625,-86.142015625,1.95940771484375],[0.000687502564593619,0.0161290141827085,0.042580986650659,-0.998962582791555],[0,0,0,0],[8.999999E+09,8.999999E+09,8.999999E+09,8.999999E+09,8.999999E+09,8.999999E+09]];
    LOCAL CONST Robtarget Tr_meulage_motif_2_150 := [[92.814,-85.1727890625,1.94912243652344],[0.000687502564593619,0.0161290141827085,0.042580986650659,-0.998962582791555],[0,0,0,0],[8.999999E+09,8.999999E+09,8.999999E+09,8.999999E+09,8.999999E+09,8.999999E+09]];
    LOCAL CONST Robtarget Tr_meulage_motif_2_151 := [[91.756265625,-84.3882421875,1.94079516601563],[0.000687502564593619,0.0161290141827085,0.042580986650659,-0.998962582791555],[0,0,0,0],[8.999999E+09,8.999999E+09,8.999999E+09,8.999999E+09,8.999999E+09,8.999999E+09]];
    LOCAL CONST Robtarget Tr_meulage_motif_2_152 := [[91.0529609375,-84.02209375,1.93690795898437],[0.000687502564593619,0.0161290141827085,0.042580986650659,-0.998962582791555],[0,0,0,0],[8.999999E+09,8.999999E+09,8.999999E+09,8.999999E+09,8.999999E+09,8.999999E+09]];
    LOCAL CONST Robtarget Tr_meulage_motif_2_153 := [[89.8751171875,-83.5842890625,1.93225830078125],[0.000687502564593619,0.0161290141827085,0.042580986650659,-0.998962582791555],[0,0,0,0],[8.999999E+09,8.999999E+09,8.999999E+09,8.999999E+09,8.999999E+09,8.999999E+09]];
    LOCAL CONST Robtarget Tr_meulage_motif_2_154 := [[89.0196171875,-83.356390625,1.92983679199219],[0.000687502564593619,0.0161290141827085,0.042580986650659,-0.998962582791555],[0,0,0,0],[8.999999E+09,8.999999E+09,8.999999E+09,8.999999E+09,8.999999E+09,8.999999E+09]];
    LOCAL CONST Robtarget Tr_meulage_motif_2_155 := [[88.079765625,-83.1917578125,1.9280859375],[0.000687502564593619,0.0161290141827085,0.042580986650659,-0.998962582791555],[0,0,0,0],[8.999999E+09,8.999999E+09,8.999999E+09,8.999999E+09,8.999999E+09,8.999999E+09]];
    LOCAL CONST Robtarget Tr_meulage_motif_2_156 := [[87.09446875,-83.125015625,1.92737329101562],[0.000687502564593619,0.0161290141827085,0.042580986650659,-0.998962582791555],[0,0,0,0],[8.999999E+09,8.999999E+09,8.999999E+09,8.999999E+09,8.999999E+09,8.999999E+09]];
    LOCAL CONST Robtarget Tr_meulage_motif_2_157 := [[86.0981015625,-83.0567421875,1.92664428710937],[0.000687502564593619,0.0161290141827085,0.042580986650659,-0.998962582791555],[0,0,0,0],[8.999999E+09,8.999999E+09,8.999999E+09,8.999999E+09,8.999999E+09,8.999999E+09]];
    LOCAL CONST Robtarget Tr_meulage_motif_2_158 := [[85.0990078125,-83.0992734375,1.92709069824219],[0.000687502564593619,0.0161290141827085,0.042580986650659,-0.998962582791555],[0,0,0,0],[8.999999E+09,8.999999E+09,8.999999E+09,8.999999E+09,8.999999E+09,8.999999E+09]];
    LOCAL CONST Robtarget Tr_meulage_motif_2_159 := [[84.0999140625,-83.1418046875,1.92753698730469],[0.000687502564593619,0.0161290141827085,0.042580986650659,-0.998962582791555],[0,0,0,0],[8.999999E+09,8.999999E+09,8.999999E+09,8.999999E+09,8.999999E+09,8.999999E+09]];
    LOCAL CONST Robtarget Tr_meulage_motif_2_160 := [[83.1008203125,-83.1843359375,1.9279833984375],[0.000687502564593619,0.0161290141827085,0.042580986650659,-0.998962582791555],[0,0,0,0],[8.999999E+09,8.999999E+09,8.999999E+09,8.999999E+09,8.999999E+09,8.999999E+09]];
    LOCAL CONST Robtarget Tr_meulage_motif_2_161 := [[82.10171875,-83.2268671875,1.9284296875],[0.000687502564593619,0.0161290141827085,0.042580986650659,-0.998962582791555],[0,0,0,0],[8.999999E+09,8.999999E+09,8.999999E+09,8.999999E+09,8.999999E+09,8.999999E+09]];
    LOCAL CONST Robtarget Tr_meulage_motif_2_162 := [[81.102625,-83.2693984375,1.92887609863281],[0.000687502564593619,0.0161290141827085,0.042580986650659,-0.998962582791555],[0,0,0,0],[8.999999E+09,8.999999E+09,8.999999E+09,8.999999E+09,8.999999E+09,8.999999E+09]];
    LOCAL CONST Robtarget Tr_meulage_motif_2_163 := [[80.10353125,-83.3119296875,1.92932250976563],[0.000687502564593619,0.0161290141827085,0.042580986650659,-0.998962582791555],[0,0,0,0],[8.999999E+09,8.999999E+09,8.999999E+09,8.999999E+09,8.999999E+09,8.999999E+09]];
    LOCAL CONST Robtarget Tr_meulage_motif_2_164 := [[79.1044375,-83.3544609375,1.92976879882813],[0.000687502564593619,0.0161290141827085,0.042580986650659,-0.998962582791555],[0,0,0,0],[8.999999E+09,8.999999E+09,8.999999E+09,8.999999E+09,8.999999E+09,8.999999E+09]];
    LOCAL CONST Robtarget Tr_meulage_motif_2_165 := [[78.10534375,-83.3969921875,1.93021520996094],[0.000687502564593619,0.0161290141827085,0.042580986650659,-0.998962582791555],[0,0,0,0],[8.999999E+09,8.999999E+09,8.999999E+09,8.999999E+09,8.999999E+09,8.999999E+09]];
    LOCAL CONST Robtarget Tr_meulage_motif_2_166 := [[77.10625,-83.4395234375,1.93066149902344],[0.000687502564593619,0.0161290141827085,0.042580986650659,-0.998962582791555],[0,0,0,0],[8.999999E+09,8.999999E+09,8.999999E+09,8.999999E+09,8.999999E+09,8.999999E+09]];
    LOCAL CONST Robtarget Tr_meulage_motif_2_167 := [[76.10715625,-83.4820546875,1.93110791015625],[0.000687502564593619,0.0161290141827085,0.042580986650659,-0.998962582791555],[0,0,0,0],[8.999999E+09,8.999999E+09,8.999999E+09,8.999999E+09,8.999999E+09,8.999999E+09]];
    LOCAL CONST Robtarget Tr_meulage_motif_2_168 := [[75.1080546875,-83.5245859375,1.93155432128906],[0.000687502564593619,0.0161290141827085,0.042580986650659,-0.998962582791555],[0,0,0,0],[8.999999E+09,8.999999E+09,8.999999E+09,8.999999E+09,8.999999E+09,8.999999E+09]];
    LOCAL CONST Robtarget Tr_meulage_motif_2_169 := [[74.1089609375,-83.5671171875,1.93200061035156],[0.000687502564593619,0.0161290141827085,0.042580986650659,-0.998962582791555],[0,0,0,0],[8.999999E+09,8.999999E+09,8.999999E+09,8.999999E+09,8.999999E+09,8.999999E+09]];
    LOCAL CONST Robtarget Tr_meulage_motif_2_170 := [[73.1098671875,-83.6096484375,1.93244702148437],[0.000687502564593619,0.0161290141827085,0.042580986650659,-0.998962582791555],[0,0,0,0],[8.999999E+09,8.999999E+09,8.999999E+09,8.999999E+09,8.999999E+09,8.999999E+09]];
    LOCAL CONST Robtarget Tr_meulage_motif_2_171 := [[72.1107734375,-83.6521796875,1.93289331054688],[0.000687502564593619,0.0161290141827085,0.042580986650659,-0.998962582791555],[0,0,0,0],[8.999999E+09,8.999999E+09,8.999999E+09,8.999999E+09,8.999999E+09,8.999999E+09]];
    LOCAL CONST Robtarget Tr_meulage_motif_2_172 := [[71.1116796875,-83.6947109375,1.93333972167969],[0.000687502564593619,0.0161290141827085,0.042580986650659,-0.998962582791555],[0,0,0,0],[8.999999E+09,8.999999E+09,8.999999E+09,8.999999E+09,8.999999E+09,8.999999E+09]];
    LOCAL CONST Robtarget Tr_meulage_motif_2_173 := [[70.1125859375,-83.73725,1.9337861328125],[0.000687502564593619,0.0161290141827085,0.042580986650659,-0.998962582791555],[0,0,0,0],[8.999999E+09,8.999999E+09,8.999999E+09,8.999999E+09,8.999999E+09,8.999999E+09]];
    LOCAL CONST Robtarget Tr_meulage_motif_2_174 := [[69.113484375,-83.77978125,1.934232421875],[0.000687502564593619,0.0161290141827085,0.042580986650659,-0.998962582791555],[0,0,0,0],[8.999999E+09,8.999999E+09,8.999999E+09,8.999999E+09,8.999999E+09,8.999999E+09]];
    LOCAL CONST Robtarget Tr_meulage_motif_2_175 := [[68.114390625,-83.8223125,1.93467883300781],[0.000687502564593619,0.0161290141827085,0.042580986650659,-0.998962582791555],[0,0,0,0],[8.999999E+09,8.999999E+09,8.999999E+09,8.999999E+09,8.999999E+09,8.999999E+09]];
    LOCAL CONST Robtarget Tr_meulage_motif_2_176 := [[67.115296875,-83.86484375,1.93512512207031],[0.000687502564593619,0.0161290141827085,0.042580986650659,-0.998962582791555],[0,0,0,0],[8.999999E+09,8.999999E+09,8.999999E+09,8.999999E+09,8.999999E+09,8.999999E+09]];
    LOCAL CONST Robtarget Tr_meulage_motif_2_177 := [[66.116203125,-83.907375,1.93557153320313],[0.000687502564593619,0.0161290141827085,0.042580986650659,-0.998962582791555],[0,0,0,0],[8.999999E+09,8.999999E+09,8.999999E+09,8.999999E+09,8.999999E+09,8.999999E+09]];
    LOCAL CONST Robtarget Tr_meulage_motif_2_178 := [[65.11710546875,-83.94990625,1.93601794433594],[0.000687502564593619,0.0161290141827085,0.042580986650659,-0.998962582791555],[0,0,0,0],[8.999999E+09,8.999999E+09,8.999999E+09,8.999999E+09,8.999999E+09,8.999999E+09]];
    LOCAL CONST Robtarget Tr_meulage_motif_2_179 := [[64.11801171875,-83.9924375,1.93646423339844],[0.000687502564593619,0.0161290141827085,0.042580986650659,-0.998962582791555],[0,0,0,0],[8.999999E+09,8.999999E+09,8.999999E+09,8.999999E+09,8.999999E+09,8.999999E+09]];
    LOCAL CONST Robtarget Tr_meulage_motif_2_180 := [[63.11891796875,-84.03496875,1.93691064453125],[0.000687502564593619,0.0161290141827085,0.042580986650659,-0.998962582791555],[0,0,0,0],[8.999999E+09,8.999999E+09,8.999999E+09,8.999999E+09,8.999999E+09,8.999999E+09]];
    LOCAL CONST Robtarget Tr_meulage_motif_2_181 := [[62.1198203125,-84.0775,1.93735693359375],[0.000687502564593619,0.0161290141827085,0.042580986650659,-0.998962582791555],[0,0,0,0],[8.999999E+09,8.999999E+09,8.999999E+09,8.999999E+09,8.999999E+09,8.999999E+09]];
    LOCAL CONST Robtarget Tr_meulage_motif_2_182 := [[61.1207265625,-84.12003125,1.93780334472656],[0.000687502564593619,0.0161290141827085,0.042580986650659,-0.998962582791555],[0,0,0,0],[8.999999E+09,8.999999E+09,8.999999E+09,8.999999E+09,8.999999E+09,8.999999E+09]];
    LOCAL CONST Robtarget Tr_meulage_motif_2_183 := [[60.1216328125,-84.1625625,1.93824975585937],[0.000687502564593619,0.0161290141827085,0.042580986650659,-0.998962582791555],[0,0,0,0],[8.999999E+09,8.999999E+09,8.999999E+09,8.999999E+09,8.999999E+09,8.999999E+09]];
    LOCAL CONST Robtarget Tr_meulage_motif_2_184 := [[59.12253515625,-84.20509375,1.93869604492188],[0.000687502564593619,0.0161290141827085,0.042580986650659,-0.998962582791555],[0,0,0,0],[8.999999E+09,8.999999E+09,8.999999E+09,8.999999E+09,8.999999E+09,8.999999E+09]];
    LOCAL CONST Robtarget Tr_meulage_motif_2_185 := [[58.12344140625,-84.247625,1.93914245605469],[0.000687502564593619,0.0161290141827085,0.042580986650659,-0.998962582791555],[0,0,0,0],[8.999999E+09,8.999999E+09,8.999999E+09,8.999999E+09,8.999999E+09,8.999999E+09]];
    LOCAL CONST Robtarget Tr_meulage_motif_2_186 := [[57.12434765625,-84.29015625,1.93958874511719],[0.000687502564593619,0.0161290141827085,0.042580986650659,-0.998962582791555],[0,0,0,0],[8.999999E+09,8.999999E+09,8.999999E+09,8.999999E+09,8.999999E+09,8.999999E+09]];
    LOCAL CONST Robtarget Tr_meulage_motif_2_187 := [[56.12525,-84.3326875,1.94003515625],[0.000687502564593619,0.0161290141827085,0.042580986650659,-0.998962582791555],[0,0,0,0],[8.999999E+09,8.999999E+09,8.999999E+09,8.999999E+09,8.999999E+09,8.999999E+09]];
    LOCAL CONST Robtarget Tr_meulage_motif_2_188 := [[55.1288828125,-84.2644140625,1.93930615234375],[0.000687502564593619,0.0161290141827085,0.042580986650659,-0.998962582791555],[0,0,0,0],[8.999999E+09,8.999999E+09,8.999999E+09,8.999999E+09,8.999999E+09,8.999999E+09]];
    LOCAL CONST Robtarget Tr_meulage_motif_2_189 := [[54.1742578125,-84.0936875,1.93749060058594],[0.000687502564593619,0.0161290141827085,0.042580986650659,-0.998962582791555],[0,0,0,0],[8.999999E+09,8.999999E+09,8.999999E+09,8.999999E+09,8.999999E+09,8.999999E+09]];
    LOCAL CONST Robtarget Tr_meulage_motif_2_190 := [[53.31074609375,-83.8583671875,1.93499035644531],[0.000687502564593619,0.0161290141827085,0.042580986650659,-0.998962582791555],[0,0,0,0],[8.999999E+09,8.999999E+09,8.999999E+09,8.999999E+09,8.999999E+09,8.999999E+09]];
    LOCAL CONST Robtarget Tr_meulage_motif_2_191 := [[52.58695703125,-83.58478125,1.93208483886719],[0.000687502564593619,0.0161290141827085,0.042580986650659,-0.998962582791555],[0,0,0,0],[8.999999E+09,8.999999E+09,8.999999E+09,8.999999E+09,8.999999E+09,8.999999E+09]];
    LOCAL CONST Robtarget Tr_meulage_motif_2_192 := [[51.5252421875,-82.9668828125,1.92552551269531],[0.000687502564593619,0.0161290141827085,0.042580986650659,-0.998962582791555],[0,0,0,0],[8.999999E+09,8.999999E+09,8.999999E+09,8.999999E+09,8.999999E+09,8.999999E+09]];
    LOCAL CONST Robtarget Tr_meulage_motif_2_193 := [[50.5857578125,-82.1041640625,1.91636962890625],[0.000687502564593619,0.0161290141827085,0.042580986650659,-0.998962582791555],[0,0,0,0],[8.999999E+09,8.999999E+09,8.999999E+09,8.999999E+09,8.999999E+09,8.999999E+09]];
    LOCAL CONST Robtarget Tr_meulage_motif_2_194 := [[50.00678125,-81.08190625,1.90552331542969],[0.000687502564593619,0.0161290141827085,0.042580986650659,-0.998962582791555],[0,0,0,0],[8.999999E+09,8.999999E+09,8.999999E+09,8.999999E+09,8.999999E+09,8.999999E+09]];
    LOCAL CONST Robtarget Tr_meulage_motif_2_195 := [[49.79268359375,-80.3971953125,1.89825927734375],[0.000687502564593619,0.0161290141827085,0.042580986650659,-0.998962582791555],[0,0,0,0],[8.999999E+09,8.999999E+09,8.999999E+09,8.999999E+09,8.999999E+09,8.999999E+09]];
    LOCAL CONST Robtarget Tr_meulage_motif_2_196 := [[49.69614453125,-79.6306484375,1.89012768554687],[0.000687502564593619,0.0161290141827085,0.042580986650659,-0.998962582791555],[0,0,0,0],[8.999999E+09,8.999999E+09,8.999999E+09,8.999999E+09,8.999999E+09,8.999999E+09]];
    LOCAL CONST Robtarget Tr_meulage_motif_2_197 := [[49.73027734375,-78.8586796875,1.88193933105469],[0.000687502564593619,0.0161290141827085,0.042580986650659,-0.998962582791555],[0,0,0,0],[8.999999E+09,8.999999E+09,8.999999E+09,8.999999E+09,8.999999E+09,8.999999E+09]];
    LOCAL CONST Robtarget Tr_meulage_motif_2_198 := [[50.10235546875,-77.73365625,1.87000732421875],[0.000687502564593619,0.0161290141827085,0.042580986650659,-0.998962582791555],[0,0,0,0],[8.999999E+09,8.999999E+09,8.999999E+09,8.999999E+09,8.999999E+09,8.999999E+09]];
    LOCAL CONST Robtarget Tr_meulage_motif_2_199 := [[50.49137890625,-77.13090625,1.86361560058594],[0.000687502564593619,0.0161290141827085,0.042580986650659,-0.998962582791555],[0,0,0,0],[8.999999E+09,8.999999E+09,8.999999E+09,8.999999E+09,8.999999E+09,8.999999E+09]];
    LOCAL CONST Robtarget Tr_meulage_motif_2_200 := [[51.33996875,-76.206875,1.85381799316406],[0.000687502564593619,0.0161290141827085,0.042580986650659,-0.998962582791555],[0,0,0,0],[8.999999E+09,8.999999E+09,8.999999E+09,8.999999E+09,8.999999E+09,8.999999E+09]];
    LOCAL CONST Robtarget Tr_meulage_motif_2_201 := [[51.90750390625,-75.768078125,1.84916625976563],[0.000687502564593619,0.0161290141827085,0.042580986650659,-0.998962582791555],[0,0,0,0],[8.999999E+09,8.999999E+09,8.999999E+09,8.999999E+09,8.999999E+09,8.999999E+09]];
    LOCAL CONST Robtarget Tr_meulage_motif_2_202 := [[53.00125390625,-75.1769296875,1.84290087890625],[0.000687502564593619,0.0161290141827085,0.042580986650659,-0.998962582791555],[0,0,0,0],[8.999999E+09,8.999999E+09,8.999999E+09,8.999999E+09,8.999999E+09,8.999999E+09]];
    LOCAL CONST Robtarget Tr_meulage_motif_2_203 := [[53.81353125,-74.8466015625,1.83940087890625],[0.000687502564593619,0.0161290141827085,0.042580986650659,-0.998962582791555],[0,0,0,0],[8.999999E+09,8.999999E+09,8.999999E+09,8.999999E+09,8.999999E+09,8.999999E+09]];
    LOCAL CONST Robtarget Tr_meulage_motif_2_204 := [[54.7359921875,-74.602671875,1.83681787109375],[0.000687502564593619,0.0161290141827085,0.042580986650659,-0.998962582791555],[0,0,0,0],[8.999999E+09,8.999999E+09,8.999999E+09,8.999999E+09,8.999999E+09,8.999999E+09]];
    LOCAL CONST Robtarget Tr_meulage_motif_2_205 := [[55.71205078125,-74.452484375,1.83522937011719],[0.000687502564593619,0.0161290141827085,0.042580986650659,-0.998962582791555],[0,0,0,0],[8.999999E+09,8.999999E+09,8.999999E+09,8.999999E+09,8.999999E+09,8.999999E+09]];
    LOCAL CONST Robtarget Tr_meulage_motif_2_206 := [[56.6990078125,-74.299765625,1.83361413574219],[0.000687502564593619,0.0161290141827085,0.042580986650659,-0.998962582791555],[0,0,0,0],[8.999999E+09,8.999999E+09,8.999999E+09,8.999999E+09,8.999999E+09,8.999999E+09]];
    LOCAL CONST Robtarget Tr_meulage_motif_2_207 := [[57.69810546875,-74.257234375,1.83316784667969],[0.000687502564593619,0.0161290141827085,0.042580986650659,-0.998962582791555],[0,0,0,0],[8.999999E+09,8.999999E+09,8.999999E+09,8.999999E+09,8.999999E+09,8.999999E+09]];
    LOCAL CONST Robtarget Tr_meulage_motif_2_208 := [[58.69719921875,-74.214703125,1.83272143554688],[0.000687502564593619,0.0161290141827085,0.042580986650659,-0.998962582791555],[0,0,0,0],[8.999999E+09,8.999999E+09,8.999999E+09,8.999999E+09,8.999999E+09,8.999999E+09]];
    LOCAL CONST Robtarget Tr_meulage_motif_2_209 := [[59.69629296875,-74.172171875,1.83227502441406],[0.000687502564593619,0.0161290141827085,0.042580986650659,-0.998962582791555],[0,0,0,0],[8.999999E+09,8.999999E+09,8.999999E+09,8.999999E+09,8.999999E+09,8.999999E+09]];
    LOCAL CONST Robtarget Tr_meulage_motif_2_210 := [[60.695390625,-74.129640625,1.83182873535156],[0.000687502564593619,0.0161290141827085,0.042580986650659,-0.998962582791555],[0,0,0,0],[8.999999E+09,8.999999E+09,8.999999E+09,8.999999E+09,8.999999E+09,8.999999E+09]];
    LOCAL CONST Robtarget Tr_meulage_motif_2_211 := [[61.694484375,-74.087109375,1.83138232421875],[0.000687502564593619,0.0161290141827085,0.042580986650659,-0.998962582791555],[0,0,0,0],[8.999999E+09,8.999999E+09,8.999999E+09,8.999999E+09,8.999999E+09,8.999999E+09]];
    LOCAL CONST Robtarget Tr_meulage_motif_2_212 := [[62.693578125,-74.044578125,1.83093603515625],[0.000687502564593619,0.0161290141827085,0.042580986650659,-0.998962582791555],[0,0,0,0],[8.999999E+09,8.999999E+09,8.999999E+09,8.999999E+09,8.999999E+09,8.999999E+09]];
    LOCAL CONST Robtarget Tr_meulage_motif_2_213 := [[63.69267578125,-74.002046875,1.83048962402344],[0.000687502564593619,0.0161290141827085,0.042580986650659,-0.998962582791555],[0,0,0,0],[8.999999E+09,8.999999E+09,8.999999E+09,8.999999E+09,8.999999E+09,8.999999E+09]];
    LOCAL CONST Robtarget Tr_meulage_motif_2_214 := [[64.69176953125,-73.959515625,1.83004321289062],[0.000687502564593619,0.0161290141827085,0.042580986650659,-0.998962582791555],[0,0,0,0],[8.999999E+09,8.999999E+09,8.999999E+09,8.999999E+09,8.999999E+09,8.999999E+09]];
    LOCAL CONST Robtarget Tr_meulage_motif_2_215 := [[65.6908671875,-73.916984375,1.82959692382813],[0.000687502564593619,0.0161290141827085,0.042580986650659,-0.998962582791555],[0,0,0,0],[8.999999E+09,8.999999E+09,8.999999E+09,8.999999E+09,8.999999E+09,8.999999E+09]];
    LOCAL CONST Robtarget Tr_meulage_motif_2_216 := [[66.6899609375,-73.874453125,1.82915051269531],[0.000687502564593619,0.0161290141827085,0.042580986650659,-0.998962582791555],[0,0,0,0],[8.999999E+09,8.999999E+09,8.999999E+09,8.999999E+09,8.999999E+09,8.999999E+09]];
    LOCAL CONST Robtarget Tr_meulage_motif_2_217 := [[67.6890546875,-73.831921875,1.82870422363281],[0.000687502564593619,0.0161290141827085,0.042580986650659,-0.998962582791555],[0,0,0,0],[8.999999E+09,8.999999E+09,8.999999E+09,8.999999E+09,8.999999E+09,8.999999E+09]];
    LOCAL CONST Robtarget Tr_meulage_motif_2_218 := [[68.6881484375,-73.789390625,1.8282578125],[0.000687502564593619,0.0161290141827085,0.042580986650659,-0.998962582791555],[0,0,0,0],[8.999999E+09,8.999999E+09,8.999999E+09,8.999999E+09,8.999999E+09,8.999999E+09]];
    LOCAL CONST Robtarget Tr_meulage_motif_2_219 := [[69.6872421875,-73.746859375,1.82781140136719],[0.000687502564593619,0.0161290141827085,0.042580986650659,-0.998962582791555],[0,0,0,0],[8.999999E+09,8.999999E+09,8.999999E+09,8.999999E+09,8.999999E+09,8.999999E+09]];
    LOCAL CONST Robtarget Tr_meulage_motif_2_220 := [[70.6863359375,-73.704328125,1.82736511230469],[0.000687502564593619,0.0161290141827085,0.042580986650659,-0.998962582791555],[0,0,0,0],[8.999999E+09,8.999999E+09,8.999999E+09,8.999999E+09,8.999999E+09,8.999999E+09]];
    LOCAL CONST Robtarget Tr_meulage_motif_2_221 := [[71.6854375,-73.661796875,1.82691870117188],[0.000687502564593619,0.0161290141827085,0.042580986650659,-0.998962582791555],[0,0,0,0],[8.999999E+09,8.999999E+09,8.999999E+09,8.999999E+09,8.999999E+09,8.999999E+09]];
    LOCAL CONST Robtarget Tr_meulage_motif_2_222 := [[72.68453125,-73.619265625,1.82647241210937],[0.000687502564593619,0.0161290141827085,0.042580986650659,-0.998962582791555],[0,0,0,0],[8.999999E+09,8.999999E+09,8.999999E+09,8.999999E+09,8.999999E+09,8.999999E+09]];
    LOCAL CONST Robtarget Tr_meulage_motif_2_223 := [[73.683625,-73.576734375,1.82602600097656],[0.000687502564593619,0.0161290141827085,0.042580986650659,-0.998962582791555],[0,0,0,0],[8.999999E+09,8.999999E+09,8.999999E+09,8.999999E+09,8.999999E+09,8.999999E+09]];
    LOCAL CONST Robtarget Tr_meulage_motif_2_224 := [[74.68271875,-73.534203125,1.82557958984375],[0.000687502564593619,0.0161290141827085,0.042580986650659,-0.998962582791555],[0,0,0,0],[8.999999E+09,8.999999E+09,8.999999E+09,8.999999E+09,8.999999E+09,8.999999E+09]];
    LOCAL CONST Robtarget Tr_meulage_motif_2_225 := [[75.6818125,-73.491671875,1.82513330078125],[0.000687502564593619,0.0161290141827085,0.042580986650659,-0.998962582791555],[0,0,0,0],[8.999999E+09,8.999999E+09,8.999999E+09,8.999999E+09,8.999999E+09,8.999999E+09]];
    LOCAL CONST Robtarget Tr_meulage_motif_2_226 := [[76.68090625,-73.449140625,1.82468688964844],[0.000687502564593619,0.0161290141827085,0.042580986650659,-0.998962582791555],[0,0,0,0],[8.999999E+09,8.999999E+09,8.999999E+09,8.999999E+09,8.999999E+09,8.999999E+09]];
    LOCAL CONST Robtarget Tr_meulage_motif_2_227 := [[77.6800078125,-73.406609375,1.82424060058594],[0.000687502564593619,0.0161290141827085,0.042580986650659,-0.998962582791555],[0,0,0,0],[8.999999E+09,8.999999E+09,8.999999E+09,8.999999E+09,8.999999E+09,8.999999E+09]];
    LOCAL CONST Robtarget Tr_meulage_motif_2_228 := [[78.6791015625,-73.364078125,1.82379418945313],[0.000687502564593619,0.0161290141827085,0.042580986650659,-0.998962582791555],[0,0,0,0],[8.999999E+09,8.999999E+09,8.999999E+09,8.999999E+09,8.999999E+09,8.999999E+09]];
    LOCAL CONST Robtarget Tr_meulage_motif_2_229 := [[79.6781953125,-73.321546875,1.82334777832031],[0.000687502564593619,0.0161290141827085,0.042580986650659,-0.998962582791555],[0,0,0,0],[8.999999E+09,8.999999E+09,8.999999E+09,8.999999E+09,8.999999E+09,8.999999E+09]];
    LOCAL CONST Robtarget Tr_meulage_motif_2_230 := [[80.6772890625,-73.279015625,1.82290148925781],[0.000687502564593619,0.0161290141827085,0.042580986650659,-0.998962582791555],[0,0,0,0],[8.999999E+09,8.999999E+09,8.999999E+09,8.999999E+09,8.999999E+09,8.999999E+09]];
    LOCAL CONST Robtarget Tr_meulage_motif_2_231 := [[81.6763828125,-73.236484375,1.822455078125],[0.000687502564593619,0.0161290141827085,0.042580986650659,-0.998962582791555],[0,0,0,0],[8.999999E+09,8.999999E+09,8.999999E+09,8.999999E+09,8.999999E+09,8.999999E+09]];
    LOCAL CONST Robtarget Tr_meulage_motif_2_232 := [[82.6754765625,-73.1939453125,1.8220087890625],[0.000687502564593619,0.0161290141827085,0.042580986650659,-0.998962582791555],[0,0,0,0],[8.999999E+09,8.999999E+09,8.999999E+09,8.999999E+09,8.999999E+09,8.999999E+09]];
    LOCAL CONST Robtarget Tr_meulage_motif_2_233 := [[83.674578125,-73.1514140625,1.82156237792969],[0.000687502564593619,0.0161290141827085,0.042580986650659,-0.998962582791555],[0,0,0,0],[8.999999E+09,8.999999E+09,8.999999E+09,8.999999E+09,8.999999E+09,8.999999E+09]];
    LOCAL CONST Robtarget Tr_meulage_motif_2_234 := [[84.673671875,-73.1088828125,1.82111596679688],[0.000687502564593619,0.0161290141827085,0.042580986650659,-0.998962582791555],[0,0,0,0],[8.999999E+09,8.999999E+09,8.999999E+09,8.999999E+09,8.999999E+09,8.999999E+09]];
    LOCAL CONST Robtarget Tr_meulage_motif_2_235 := [[85.672765625,-73.0663515625,1.82066967773437],[0.000687502564593619,0.0161290141827085,0.042580986650659,-0.998962582791555],[0,0,0,0],[8.999999E+09,8.999999E+09,8.999999E+09,8.999999E+09,8.999999E+09,8.999999E+09]];
    LOCAL CONST Robtarget Tr_meulage_motif_2_236 := [[86.671859375,-73.0238203125,1.82022326660156],[0.000687502564593619,0.0161290141827085,0.042580986650659,-0.998962582791555],[0,0,0,0],[8.999999E+09,8.999999E+09,8.999999E+09,8.999999E+09,8.999999E+09,8.999999E+09]];
    LOCAL CONST Robtarget Tr_meulage_motif_2_237 := [[87.6588203125,-72.8711015625,1.81860803222656],[0.000687502564593619,0.0161290141827085,0.042580986650659,-0.998962582791555],[0,0,0,0],[8.999999E+09,8.999999E+09,8.999999E+09,8.999999E+09,8.999999E+09,8.999999E+09]];
    LOCAL CONST Robtarget Tr_meulage_motif_2_238 := [[88.5954765625,-72.6198671875,1.81594750976563],[0.000687502564593619,0.0161290141827085,0.042580986650659,-0.998962582791555],[0,0,0,0],[8.999999E+09,8.999999E+09,8.999999E+09,8.999999E+09,8.999999E+09,8.999999E+09]];
    LOCAL CONST Robtarget Tr_meulage_motif_2_239 := [[89.4358671875,-72.31203125,1.81268627929687],[0.000687502564593619,0.0161290141827085,0.042580986650659,-0.998962582791555],[0,0,0,0],[8.999999E+09,8.999999E+09,8.999999E+09,8.999999E+09,8.999999E+09,8.999999E+09]];
    LOCAL CONST Robtarget Tr_meulage_motif_2_240 := [[90.1337890625,-71.977921875,1.8091455078125],[0.000687502564593619,0.0161290141827085,0.042580986650659,-0.998962582791555],[0,0,0,0],[8.999999E+09,8.999999E+09,8.999999E+09,8.999999E+09,8.999999E+09,8.999999E+09]];
    LOCAL CONST Robtarget Tr_meulage_motif_2_241 := [[91.139140625,-71.27203125,1.80166259765625],[0.000687502564593619,0.0161290141827085,0.042580986650659,-0.998962582791555],[0,0,0,0],[8.999999E+09,8.999999E+09,8.999999E+09,8.999999E+09,8.999999E+09,8.999999E+09]];
    LOCAL CONST Robtarget Tr_meulage_motif_2_242 := [[91.9113046875,-70.298578125,1.79134045410156],[0.000687502564593619,0.0161290141827085,0.042580986650659,-0.998962582791555],[0,0,0,0],[8.999999E+09,8.999999E+09,8.999999E+09,8.999999E+09,8.999999E+09,8.999999E+09]];
    LOCAL CONST Robtarget Tr_meulage_motif_2_243 := [[92.221046875,-69.2881875,1.78062426757812],[0.000687502564593619,0.0161290141827085,0.042580986650659,-0.998962582791555],[0,0,0,0],[8.999999E+09,8.999999E+09,8.999999E+09,8.999999E+09,8.999999E+09,8.999999E+09]];
    LOCAL CONST Robtarget Tr_meulage_motif_2_244 := [[92.167703125,-68.7324375,1.77472888183594],[0.000687502564593619,0.0161290141827085,0.042580986650659,-0.998962582791555],[0,0,0,0],[8.999999E+09,8.999999E+09,8.999999E+09,8.999999E+09,8.999999E+09,8.999999E+09]];
    LOCAL CONST Robtarget Tr_meulage_motif_2_245 := [[92.154234375,-68.31475,1.77029821777344],[0.000687502564593619,0.0161290141827085,0.042580986650659,-0.998962582791555],[0,0,0,0],[8.999999E+09,8.999999E+09,8.999999E+09,8.999999E+09,8.999999E+09,8.999999E+09]];
    LOCAL CONST Robtarget Tr_meulage_motif_2_246 := [[91.7511796875,-67.3617578125,1.7601875],[0.000687502564593619,0.0161290141827085,0.042580986650659,-0.998962582791555],[0,0,0,0],[8.999999E+09,8.999999E+09,8.999999E+09,8.999999E+09,8.999999E+09,8.999999E+09]];
    LOCAL CONST Robtarget Tr_meulage_motif_2_247 := [[90.890953125,-66.47990625,1.75082922363281],[0.000687502564593619,0.0161290141827085,0.042580986650659,-0.998962582791555],[0,0,0,0],[8.999999E+09,8.999999E+09,8.999999E+09,8.999999E+09,8.999999E+09,8.999999E+09]];
    LOCAL CONST Robtarget Tr_meulage_motif_2_248 := [[90.261359375,-66.0834609375,1.74662084960938],[0.000687502564593619,0.0161290141827085,0.042580986650659,-0.998962582791555],[0,0,0,0],[8.999999E+09,8.999999E+09,8.999999E+09,8.999999E+09,8.999999E+09,8.999999E+09]];
    LOCAL CONST Robtarget Tr_meulage_motif_2_249 := [[89.1095078125,-65.60159375,1.74150402832031],[0.000687502564593619,0.0161290141827085,0.042580986650659,-0.998962582791555],[0,0,0,0],[8.999999E+09,8.999999E+09,8.999999E+09,8.999999E+09,8.999999E+09,8.999999E+09]];
    LOCAL CONST Robtarget Tr_meulage_motif_2_250 := [[88.2540078125,-65.37367578125,1.73908227539062],[0.000687502564593619,0.0161290141827085,0.042580986650659,-0.998962582791555],[0,0,0,0],[8.999999E+09,8.999999E+09,8.999999E+09,8.999999E+09,8.999999E+09,8.999999E+09]];
    LOCAL CONST Robtarget Tr_meulage_motif_2_251 := [[87.31415625,-65.20902734375,1.73733129882813],[0.000687502564593619,0.0161290141827085,0.042580986650659,-0.998962582791555],[0,0,0,0],[8.999999E+09,8.999999E+09,8.999999E+09,8.999999E+09,8.999999E+09,8.999999E+09]];
    LOCAL CONST Robtarget Tr_meulage_motif_2_252 := [[86.3288671875,-65.14233203125,1.73661901855469],[0.000687502564593619,0.0161290141827085,0.042580986650659,-0.998962582791555],[0,0,0,0],[8.999999E+09,8.999999E+09,8.999999E+09,8.999999E+09,8.999999E+09,8.999999E+09]];
    LOCAL CONST Robtarget Tr_meulage_motif_2_253 := [[85.3324921875,-65.07404296875,1.73588989257812],[0.000687502564593619,0.0161290141827085,0.042580986650659,-0.998962582791555],[0,0,0,0],[8.999999E+09,8.999999E+09,8.999999E+09,8.999999E+09,8.999999E+09,8.999999E+09]];
    LOCAL CONST Robtarget Tr_meulage_motif_2_254 := [[84.3333984375,-65.11657421875,1.73633630371094],[0.000687502564593619,0.0161290141827085,0.042580986650659,-0.998962582791555],[0,0,0,0],[8.999999E+09,8.999999E+09,8.999999E+09,8.999999E+09,8.999999E+09,8.999999E+09]];
    LOCAL CONST Robtarget Tr_meulage_motif_2_255 := [[83.3343046875,-65.15910546875,1.73678271484375],[0.000687502564593619,0.0161290141827085,0.042580986650659,-0.998962582791555],[0,0,0,0],[8.999999E+09,8.999999E+09,8.999999E+09,8.999999E+09,8.999999E+09,8.999999E+09]];
    LOCAL CONST Robtarget Tr_meulage_motif_2_256 := [[82.3352109375,-65.20163671875,1.73722900390625],[0.000687502564593619,0.0161290141827085,0.042580986650659,-0.998962582791555],[0,0,0,0],[8.999999E+09,8.999999E+09,8.999999E+09,8.999999E+09,8.999999E+09,8.999999E+09]];
    LOCAL CONST Robtarget Tr_meulage_motif_2_257 := [[81.3361171875,-65.244171875,1.73767541503906],[0.000687502564593619,0.0161290141827085,0.042580986650659,-0.998962582791555],[0,0,0,0],[8.999999E+09,8.999999E+09,8.999999E+09,8.999999E+09,8.999999E+09,8.999999E+09]];
    LOCAL CONST Robtarget Tr_meulage_motif_2_258 := [[80.337015625,-65.286703125,1.73812170410156],[0.000687502564593619,0.0161290141827085,0.042580986650659,-0.998962582791555],[0,0,0,0],[8.999999E+09,8.999999E+09,8.999999E+09,8.999999E+09,8.999999E+09,8.999999E+09]];
    LOCAL CONST Robtarget Tr_meulage_motif_2_259 := [[79.337921875,-65.329234375,1.73856811523438],[0.000687502564593619,0.0161290141827085,0.042580986650659,-0.998962582791555],[0,0,0,0],[8.999999E+09,8.999999E+09,8.999999E+09,8.999999E+09,8.999999E+09,8.999999E+09]];
    LOCAL CONST Robtarget Tr_meulage_motif_2_260 := [[78.338828125,-65.371765625,1.73901452636719],[0.000687502564593619,0.0161290141827085,0.042580986650659,-0.998962582791555],[0,0,0,0],[8.999999E+09,8.999999E+09,8.999999E+09,8.999999E+09,8.999999E+09,8.999999E+09]];
    LOCAL CONST Robtarget Tr_meulage_motif_2_261 := [[77.339734375,-65.414296875,1.73946081542969],[0.000687502564593619,0.0161290141827085,0.042580986650659,-0.998962582791555],[0,0,0,0],[8.999999E+09,8.999999E+09,8.999999E+09,8.999999E+09,8.999999E+09,8.999999E+09]];
    LOCAL CONST Robtarget Tr_meulage_motif_2_262 := [[76.340640625,-65.456828125,1.7399072265625],[0.000687502564593619,0.0161290141827085,0.042580986650659,-0.998962582791555],[0,0,0,0],[8.999999E+09,8.999999E+09,8.999999E+09,8.999999E+09,8.999999E+09,8.999999E+09]];
    LOCAL CONST Robtarget Tr_meulage_motif_2_263 := [[75.341546875,-65.499359375,1.740353515625],[0.000687502564593619,0.0161290141827085,0.042580986650659,-0.998962582791555],[0,0,0,0],[8.999999E+09,8.999999E+09,8.999999E+09,8.999999E+09,8.999999E+09,8.999999E+09]];
    LOCAL CONST Robtarget Tr_meulage_motif_2_264 := [[74.342453125,-65.541890625,1.74079992675781],[0.000687502564593619,0.0161290141827085,0.042580986650659,-0.998962582791555],[0,0,0,0],[8.999999E+09,8.999999E+09,8.999999E+09,8.999999E+09,8.999999E+09,8.999999E+09]];
    LOCAL CONST Robtarget Tr_meulage_motif_2_265 := [[73.3433515625,-65.584421875,1.74124633789063],[0.000687502564593619,0.0161290141827085,0.042580986650659,-0.998962582791555],[0,0,0,0],[8.999999E+09,8.999999E+09,8.999999E+09,8.999999E+09,8.999999E+09,8.999999E+09]];
    LOCAL CONST Robtarget Tr_meulage_motif_2_266 := [[72.3442578125,-65.626953125,1.74169262695312],[0.000687502564593619,0.0161290141827085,0.042580986650659,-0.998962582791555],[0,0,0,0],[8.999999E+09,8.999999E+09,8.999999E+09,8.999999E+09,8.999999E+09,8.999999E+09]];
    LOCAL CONST Robtarget Tr_meulage_motif_2_267 := [[71.3451640625,-65.669484375,1.74213903808594],[0.000687502564593619,0.0161290141827085,0.042580986650659,-0.998962582791555],[0,0,0,0],[8.999999E+09,8.999999E+09,8.999999E+09,8.999999E+09,8.999999E+09,8.999999E+09]];
    LOCAL CONST Robtarget Tr_meulage_motif_2_268 := [[70.3460703125,-65.712015625,1.74258532714844],[0.000687502564593619,0.0161290141827085,0.042580986650659,-0.998962582791555],[0,0,0,0],[8.999999E+09,8.999999E+09,8.999999E+09,8.999999E+09,8.999999E+09,8.999999E+09]];
    LOCAL CONST Robtarget Tr_meulage_motif_2_269 := [[69.3469765625,-65.754546875,1.74303173828125],[0.000687502564593619,0.0161290141827085,0.042580986650659,-0.998962582791555],[0,0,0,0],[8.999999E+09,8.999999E+09,8.999999E+09,8.999999E+09,8.999999E+09,8.999999E+09]];
    LOCAL CONST Robtarget Tr_meulage_motif_2_270 := [[68.3478828125,-65.797078125,1.74347814941406],[0.000687502564593619,0.0161290141827085,0.042580986650659,-0.998962582791555],[0,0,0,0],[8.999999E+09,8.999999E+09,8.999999E+09,8.999999E+09,8.999999E+09,8.999999E+09]];
    LOCAL CONST Robtarget Tr_meulage_motif_2_271 := [[67.34878125,-65.839609375,1.74392443847656],[0.000687502564593619,0.0161290141827085,0.042580986650659,-0.998962582791555],[0,0,0,0],[8.999999E+09,8.999999E+09,8.999999E+09,8.999999E+09,8.999999E+09,8.999999E+09]];
    LOCAL CONST Robtarget Tr_meulage_motif_2_272 := [[66.3496875,-65.882140625,1.74437084960938],[0.000687502564593619,0.0161290141827085,0.042580986650659,-0.998962582791555],[0,0,0,0],[8.999999E+09,8.999999E+09,8.999999E+09,8.999999E+09,8.999999E+09,8.999999E+09]];
    LOCAL CONST Robtarget Tr_meulage_motif_2_273 := [[65.35059375,-65.924671875,1.74481713867187],[0.000687502564593619,0.0161290141827085,0.042580986650659,-0.998962582791555],[0,0,0,0],[8.999999E+09,8.999999E+09,8.999999E+09,8.999999E+09,8.999999E+09,8.999999E+09]];
    LOCAL CONST Robtarget Tr_meulage_motif_2_274 := [[64.3515,-65.967203125,1.74526354980469],[0.000687502564593619,0.0161290141827085,0.042580986650659,-0.998962582791555],[0,0,0,0],[8.999999E+09,8.999999E+09,8.999999E+09,8.999999E+09,8.999999E+09,8.999999E+09]];
    LOCAL CONST Robtarget Tr_meulage_motif_2_275 := [[63.35240234375,-66.009734375,1.7457099609375],[0.000687502564593619,0.0161290141827085,0.042580986650659,-0.998962582791555],[0,0,0,0],[8.999999E+09,8.999999E+09,8.999999E+09,8.999999E+09,8.999999E+09,8.999999E+09]];
    LOCAL CONST Robtarget Tr_meulage_motif_2_276 := [[62.35330859375,-66.052265625,1.74615625],[0.000687502564593619,0.0161290141827085,0.042580986650659,-0.998962582791555],[0,0,0,0],[8.999999E+09,8.999999E+09,8.999999E+09,8.999999E+09,8.999999E+09,8.999999E+09]];
    LOCAL CONST Robtarget Tr_meulage_motif_2_277 := [[61.35421484375,-66.094796875,1.74660266113281],[0.000687502564593619,0.0161290141827085,0.042580986650659,-0.998962582791555],[0,0,0,0],[8.999999E+09,8.999999E+09,8.999999E+09,8.999999E+09,8.999999E+09,8.999999E+09]];
    LOCAL CONST Robtarget Tr_meulage_motif_2_278 := [[60.3551171875,-66.137328125,1.74704895019531],[0.000687502564593619,0.0161290141827085,0.042580986650659,-0.998962582791555],[0,0,0,0],[8.999999E+09,8.999999E+09,8.999999E+09,8.999999E+09,8.999999E+09,8.999999E+09]];
    LOCAL CONST Robtarget Tr_meulage_motif_2_279 := [[59.3560234375,-66.179859375,1.74749536132812],[0.000687502564593619,0.0161290141827085,0.042580986650659,-0.998962582791555],[0,0,0,0],[8.999999E+09,8.999999E+09,8.999999E+09,8.999999E+09,8.999999E+09,8.999999E+09]];
    LOCAL CONST Robtarget Tr_meulage_motif_2_280 := [[58.3569296875,-66.222390625,1.74794177246094],[0.000687502564593619,0.0161290141827085,0.042580986650659,-0.998962582791555],[0,0,0,0],[8.999999E+09,8.999999E+09,8.999999E+09,8.999999E+09,8.999999E+09,8.999999E+09]];
    LOCAL CONST Robtarget Tr_meulage_motif_2_281 := [[57.35783203125,-66.264921875,1.74838806152344],[0.000687502564593619,0.0161290141827085,0.042580986650659,-0.998962582791555],[0,0,0,0],[8.999999E+09,8.999999E+09,8.999999E+09,8.999999E+09,8.999999E+09,8.999999E+09]];
    LOCAL CONST Robtarget Tr_meulage_motif_2_282 := [[56.35873828125,-66.307453125,1.74883447265625],[0.000687502564593619,0.0161290141827085,0.042580986650659,-0.998962582791555],[0,0,0,0],[8.999999E+09,8.999999E+09,8.999999E+09,8.999999E+09,8.999999E+09,8.999999E+09]];
    LOCAL CONST Robtarget Tr_meulage_motif_2_283 := [[55.35964453125,-66.349984375,1.74928076171875],[0.000687502564593619,0.0161290141827085,0.042580986650659,-0.998962582791555],[0,0,0,0],[8.999999E+09,8.999999E+09,8.999999E+09,8.999999E+09,8.999999E+09,8.999999E+09]];
    LOCAL CONST Robtarget Tr_meulage_motif_2_284 := [[54.360546875,-66.392515625,1.74972717285156],[0.000687502564593619,0.0161290141827085,0.042580986650659,-0.998962582791555],[0,0,0,0],[8.999999E+09,8.999999E+09,8.999999E+09,8.999999E+09,8.999999E+09,8.999999E+09]];
    LOCAL CONST Robtarget Tr_meulage_motif_2_285 := [[53.361453125,-66.435046875,1.75017358398438],[0.000687502564593619,0.0161290141827085,0.042580986650659,-0.998962582791555],[0,0,0,0],[8.999999E+09,8.999999E+09,8.999999E+09,8.999999E+09,8.999999E+09,8.999999E+09]];
    LOCAL CONST Robtarget Tr_meulage_motif_2_286 := [[52.362359375,-66.477578125,1.75061987304687],[0.000687502564593619,0.0161290141827085,0.042580986650659,-0.998962582791555],[0,0,0,0],[8.999999E+09,8.999999E+09,8.999999E+09,8.999999E+09,8.999999E+09,8.999999E+09]];
    LOCAL CONST Robtarget Tr_meulage_motif_2_287 := [[51.36326171875,-66.520109375,1.75106628417969],[0.000687502564593619,0.0161290141827085,0.042580986650659,-0.998962582791555],[0,0,0,0],[8.999999E+09,8.999999E+09,8.999999E+09,8.999999E+09,8.999999E+09,8.999999E+09]];
    LOCAL CONST Robtarget Tr_meulage_motif_2_288 := [[50.36416796875,-66.5626484375,1.75151257324219],[0.000687502564593619,0.0161290141827085,0.042580986650659,-0.998962582791555],[0,0,0,0],[8.999999E+09,8.999999E+09,8.999999E+09,8.999999E+09,8.999999E+09,8.999999E+09]];
    LOCAL CONST Robtarget Tr_meulage_motif_2_289 := [[49.36507421875,-66.6051796875,1.751958984375],[0.000687502564593619,0.0161290141827085,0.042580986650659,-0.998962582791555],[0,0,0,0],[8.999999E+09,8.999999E+09,8.999999E+09,8.999999E+09,8.999999E+09,8.999999E+09]];
    LOCAL CONST Robtarget Tr_meulage_motif_2_290 := [[48.3659765625,-66.6477109375,1.75240539550781],[0.000687502564593619,0.0161290141827085,0.042580986650659,-0.998962582791555],[0,0,0,0],[8.999999E+09,8.999999E+09,8.999999E+09,8.999999E+09,8.999999E+09,8.999999E+09]];
    LOCAL CONST Robtarget Tr_meulage_motif_2_291 := [[47.3668828125,-66.6902421875,1.75285168457031],[0.000687502564593619,0.0161290141827085,0.042580986650659,-0.998962582791555],[0,0,0,0],[8.999999E+09,8.999999E+09,8.999999E+09,8.999999E+09,8.999999E+09,8.999999E+09]];
    LOCAL CONST Robtarget Tr_meulage_motif_2_292 := [[46.3677890625,-66.7327734375,1.75329809570313],[0.000687502564593619,0.0161290141827085,0.042580986650659,-0.998962582791555],[0,0,0,0],[8.999999E+09,8.999999E+09,8.999999E+09,8.999999E+09,8.999999E+09,8.999999E+09]];
    LOCAL CONST Robtarget Tr_meulage_motif_2_293 := [[45.3686953125,-66.7753046875,1.75374438476563],[0.000687502564593619,0.0161290141827085,0.042580986650659,-0.998962582791555],[0,0,0,0],[8.999999E+09,8.999999E+09,8.999999E+09,8.999999E+09,8.999999E+09,8.999999E+09]];
    LOCAL CONST Robtarget Tr_meulage_motif_2_294 := [[44.36959765625,-66.8178359375,1.75419079589844],[0.000687502564593619,0.0161290141827085,0.042580986650659,-0.998962582791555],[0,0,0,0],[8.999999E+09,8.999999E+09,8.999999E+09,8.999999E+09,8.999999E+09,8.999999E+09]];

